LIN {X 0,Y 418.254,Z 60.388,A -85,B 0,C 180,E1 -10209.681,E2 -10209.681} C_VEL
LIN {X 0,Y 418.228,Z 60.388,A -85,B 0,C 180,E1 -10212.321,E2 -10212.321} C_VEL
LIN {X 0,Y 418.234,Z 60.379,A -85,B 0,C 180,E1 -10215.108,E2 -10215.108} C_VEL
LIN {X 0,Y 418.254,Z 60.387,A -85,B 0,C 180,E1 -10217.769,E2 -10217.769} C_VEL
LIN {X 0,Y 418.266,Z 60.381,A -85,B 0,C 180,E1 -10220.616,E2 -10220.616} C_VEL
LIN {X 0,Y 418.244,Z 60.385,A -85,B 0,C 180,E1 -10223.976,E2 -10223.976} C_VEL
LIN {X 0,Y 418.255,Z 60.388,A -85,B 0,C 180,E1 -10227.156,E2 -10227.156} C_VEL
LIN {X 0,Y 418.266,Z 60.385,A -85,B 0,C 180,E1 -10230.895,E2 -10230.895} C_VEL
LIN {X 0,Y 418.269,Z 60.378,A -85,B 0,C 180,E1 -10234.096,E2 -10234.096} C_VEL
LIN {X 0,Y 418.236,Z 60.379,A -85,B 0,C 180,E1 -10237.264,E2 -10237.264} C_VEL
LIN {X 0,Y 418.314,Z 60.38,A -85,B 0,C 180,E1 -10240.366,E2 -10240.366} C_VEL
LIN {X 0,Y 418.315,Z 60.373,A -85,B 0,C 180,E1 -10243.405,E2 -10243.405} C_VEL
LIN {X 0,Y 418.343,Z 60.364,A -85,B 0,C 180,E1 -10246.999,E2 -10246.999} C_VEL
LIN {X 0,Y 418.355,Z 60.373,A -85,B 0,C 180,E1 -10250.329,E2 -10250.329} C_VEL
LIN {X 0,Y 418.485,Z 60.349,A -85,B 0,C 180,E1 -10253.249,E2 -10253.249} C_VEL
LIN {X 0,Y 418.335,Z 60.373,A -85,B 0,C 180,E1 -10255.182,E2 -10255.182} C_VEL
LIN {X 0,Y 418.539,Z 60.345,A -85,B 0,C 180,E1 -10258.076,E2 -10258.076} C_VEL
LIN {X 0,Y 418.668,Z 60.335,A -85,B 0,C 180,E1 -10260,E2 -10260} C_VEL
LIN {X 0,Y 418.498,Z 60.346,A -85,B 0,C 180,E1 -10262.888,E2 -10262.888} C_VEL
LIN {X 0,Y 418.467,Z 60.355,A -85,B 0,C 180,E1 -10266.626,E2 -10266.626} C_VEL
LIN {X 0,Y 418.337,Z 60.376,A -85,B 0,C 180,E1 -10269.672,E2 -10269.672} C_VEL
LIN {X 0,Y 418.344,Z 60.369,A -85,B 0,C 180,E1 -10273.001,E2 -10273.001} C_VEL
LIN {X 0,Y 418.31,Z 60.378,A -85,B 0,C 180,E1 -10276.736,E2 -10276.736} C_VEL
LIN {X 0,Y 418.269,Z 60.381,A -85,B 0,C 180,E1 -10279.791,E2 -10279.791} C_VEL
LIN {X 0,Y 418.23,Z 60.386,A -85,B 0,C 180,E1 -10282.737,E2 -10282.737} C_VEL
LIN {X 0,Y 418.236,Z 60.381,A -85,B 0,C 180,E1 -10285.907,E2 -10285.907} C_VEL
LIN {X 0,Y 418.259,Z 60.38,A -85,B 0,C 180,E1 -10289.163,E2 -10289.163} C_VEL
LIN {X 0,Y 418.256,Z 60.385,A -85,B 0,C 180,E1 -10292.844,E2 -10292.844} C_VEL
LIN {X 0,Y 418.242,Z 60.39,A -85,B 0,C 180,E1 -10296.238,E2 -10296.238} C_VEL
LIN {X 0,Y 418.226,Z 60.393,A -85,B 0,C 180,E1 -10299.685,E2 -10299.685} C_VEL
LIN {X 0,Y 418.212,Z 60.393,A -85,B 0,C 180,E1 -10302.319,E2 -10302.319} C_VEL
LIN {X 0,Y 418.236,Z 60.384,A -85,B 0,C 180,E1 -10305.109,E2 -10305.109} C_VEL
LIN {X 0,Y 418.223,Z 60.394,A -85,B 0,C 180,E1 -10307.765,E2 -10307.765} C_VEL
LIN {X 0,Y 418.236,Z 60.391,A -85,B 0,C 180,E1 -10311.557,E2 -10311.557} C_VEL
LIN {X 0,Y 418.252,Z 60.396,A -85,B 0,C 180,E1 -10314.274,E2 -10314.274} C_VEL
LIN {X 0,Y 420.013,Z 68.936,A -85,B 0,C 180,E1 -10316.521,E2 -10316.521} C_VEL
LIN {X 0,Y 423.496,Z 79.315,A -85,B 0,C 180,E1 -10316.909,E2 -10316.909} C_VEL
LIN {X 0,Y 425.292,Z 87.787,A -85,B 0,C 180,E1 -10317.161,E2 -10317.161} C_VEL
LIN {X 0,Y 424.004,Z 175.768,A -85,B 0,C 180,E1 -10318.7,E2 -10318.7} C_VEL
LIN {X 0,Y 423.614,Z 189.086,A -85,B 0,C 180,E1 -10319.133,E2 -10319.133} C_VEL
LIN {X 0,Y 423.144,Z 201.473,A -85,B 0,C 180,E1 -10319.732,E2 -10319.732} C_VEL
LIN {X 0,Y 422.489,Z 212.909,A -85,B 0,C 180,E1 -10320.475,E2 -10320.475} C_VEL
LIN {X 0,Y 421.694,Z 223.677,A -85,B 0,C 180,E1 -10321.371,E2 -10321.371} C_VEL
LIN {X 0,Y 420.851,Z 234.525,A -85,B 0,C 180,E1 -10322.504,E2 -10322.504} C_VEL
LIN {X 0,Y 420.131,Z 243.656,A -85,B 0,C 180,E1 -10323.686,E2 -10323.686} C_VEL
LIN {X 0,Y 419.464,Z 251.347,A -85,B 0,C 180,E1 -10324.9,E2 -10324.9} C_VEL
LIN {X 0,Y 418.82,Z 258.37,A -85,B 0,C 180,E1 -10326.251,E2 -10326.251} C_VEL
LIN {X 0,Y 418.209,Z 265.233,A -85,B 0,C 180,E1 -10327.913,E2 -10327.913} C_VEL
LIN {X 0,Y 417.874,Z 269.767,A -85,B 0,C 180,E1 -10329.318,E2 -10329.318} C_VEL
LIN {X 0,Y 417.63,Z 272.711,A -85,B 0,C 180,E1 -10330.458,E2 -10330.458} C_VEL
LIN {X 0,Y 417.272,Z 276.201,A -85,B 0,C 180,E1 -10332.352,E2 -10332.352} C_VEL
LIN {X 0,Y 417.155,Z 277.802,A -85,B 0,C 180,E1 -10333.804,E2 -10333.804} C_VEL
LIN {X 0,Y 417.051,Z 278.53,A -85,B 0,C 180,E1 -10335.359,E2 -10335.359} C_VEL
LIN {X 0,Y 417.058,Z 278.473,A -85,B 0,C 180,E1 -10336.355,E2 -10336.355} C_VEL
LIN {X 0,Y 417.135,Z 277.669,A -85,B 0,C 180,E1 -10337.744,E2 -10337.744} C_VEL
LIN {X 0,Y 417.199,Z 275.772,A -85,B 0,C 180,E1 -10339.322,E2 -10339.322} C_VEL
LIN {X 0,Y 417.368,Z 272.99,A -85,B 0,C 180,E1 -10340.795,E2 -10340.795} C_VEL
LIN {X 0,Y 417.572,Z 269.183,A -85,B 0,C 180,E1 -10342.262,E2 -10342.262} C_VEL
LIN {X 0,Y 417.695,Z 267.355,A -85,B 0,C 180,E1 -10342.846,E2 -10342.846} C_VEL
LIN {X 0,Y 417.151,Z 264.881,A -85,B 0,C 180,E1 -10343.576,E2 -10343.576} C_VEL
LIN {X 0,Y 414.523,Z 260.479,A -85,B 0,C 180,E1 -10344.746,E2 -10344.746} C_VEL
LIN {X 0,Y 411.989,Z 255.452,A -85,B 0,C 180,E1 -10345.882,E2 -10345.882} C_VEL
LIN {X 0,Y 411.602,Z 251.956,A -85,B 0,C 180,E1 -10346.549,E2 -10346.549} C_VEL
LIN {X 0,Y 412.184,Z 244.156,A -85,B 0,C 180,E1 -10347.802,E2 -10347.802} C_VEL
LIN {X 0,Y 412.878,Z 234.823,A -85,B 0,C 180,E1 -10349.025,E2 -10349.025} C_VEL
LIN {X 0,Y 413.535,Z 224.477,A -85,B 0,C 180,E1 -10350.122,E2 -10350.122} C_VEL
LIN {X 0,Y 414.222,Z 212.979,A -85,B 0,C 180,E1 -10351.094,E2 -10351.094} C_VEL
LIN {X 0,Y 414.732,Z 200.897,A -85,B 0,C 180,E1 -10351.882,E2 -10351.882} C_VEL
LIN {X 0,Y 415.104,Z 187.886,A -85,B 0,C 180,E1 -10352.502,E2 -10352.502} C_VEL
LIN {X 0,Y 415.493,Z 174.927,A -85,B 0,C 180,E1 -10352.909,E2 -10352.909} C_VEL
LIN {X 0,Y 416.383,Z 86.513,A -85,B 0,C 180,E1 -10354.459,E2 -10354.459} C_VEL
LIN {X 0,Y 412.646,Z 68.641,A -85,B 0,C 180,E1 -10354.931,E2 -10354.931} C_VEL
LIN {X 0,Y 411.478,Z 61.231,A -85,B 0,C 180,E1 -10356.805,E2 -10356.805} C_VEL
LIN {X 0,Y 411.36,Z 61.245,A -85,B 0,C 180,E1 -10358.845,E2 -10358.845} C_VEL
LIN {X 0,Y 411.289,Z 61.25,A -85,B 0,C 180,E1 -10361.833,E2 -10361.833} C_VEL
LIN {X 0,Y 411.266,Z 61.255,A -85,B 0,C 180,E1 -10364.853,E2 -10364.853} C_VEL
LIN {X 0,Y 411.256,Z 61.256,A -85,B 0,C 180,E1 -10367.915,E2 -10367.915} C_VEL
LIN {X 0,Y 411.202,Z 61.26,A -85,B 0,C 180,E1 -10371.034,E2 -10371.034} C_VEL
LIN {X 0,Y 411.225,Z 61.263,A -85,B 0,C 180,E1 -10374.216,E2 -10374.216} C_VEL
LIN {X 0,Y 411.264,Z 61.254,A -85,B 0,C 180,E1 -10377.478,E2 -10377.478} C_VEL
LIN {X 0,Y 411.194,Z 61.261,A -85,B 0,C 180,E1 -10380.848,E2 -10380.848} C_VEL
LIN {X 0,Y 411.211,Z 61.26,A -85,B 0,C 180,E1 -10384.333,E2 -10384.333} C_VEL
LIN {X 0,Y 411.206,Z 61.263,A -85,B 0,C 180,E1 -10387.973,E2 -10387.973} C_VEL
LIN {X 0,Y 411.188,Z 61.262,A -85,B 0,C 180,E1 -10390.504,E2 -10390.504} C_VEL
LIN {X 0,Y 411.178,Z 61.267,A -85,B 0,C 180,E1 -10393.133,E2 -10393.133} C_VEL
LIN {X 0,Y 411.172,Z 61.265,A -85,B 0,C 180,E1 -10395.881,E2 -10395.881} C_VEL
LIN {X 0,Y 411.167,Z 61.266,A -85,B 0,C 180,E1 -10398.772,E2 -10398.772} C_VEL
LIN {X 0,Y 411.208,Z 61.26,A -85,B 0,C 180,E1 -10401.831,E2 -10401.831} C_VEL
LIN {X 0,Y 411.214,Z 61.264,A -85,B 0,C 180,E1 -10405.121,E2 -10405.121} C_VEL
LIN {X 0,Y 411.169,Z 61.264,A -85,B 0,C 180,E1 -10408.003,E2 -10408.003} C_VEL
LIN {X 0,Y 411.221,Z 61.259,A -85,B 0,C 180,E1 -10411.41,E2 -10411.41} C_VEL
LIN {X 0,Y 411.241,Z 61.255,A -85,B 0,C 180,E1 -10413.619,E2 -10413.619} C_VEL
LIN {X 0,Y 411.207,Z 61.264,A -85,B 0,C 180,E1 -10416.852,E2 -10416.852} C_VEL
LIN {X 0,Y 411.218,Z 61.26,A -85,B 0,C 180,E1 -10420.05,E2 -10420.05} C_VEL
LIN {X 0,Y 411.266,Z 61.253,A -85,B 0,C 180,E1 -10423.131,E2 -10423.131} C_VEL
LIN {X 0,Y 411.308,Z 61.248,A -85,B 0,C 180,E1 -10426.896,E2 -10426.896} C_VEL
LIN {X 0,Y 411.295,Z 61.255,A -85,B 0,C 180,E1 -10430.161,E2 -10430.161} C_VEL
LIN {X 0,Y 411.455,Z 61.229,A -85,B 0,C 180,E1 -10433.133,E2 -10433.133} C_VEL
LIN {X 0,Y 411.31,Z 61.247,A -85,B 0,C 180,E1 -10435.099,E2 -10435.099} C_VEL
LIN {X 0,Y 411.513,Z 61.226,A -85,B 0,C 180,E1 -10438.042,E2 -10438.042} C_VEL
LIN {X 0,Y 411.642,Z 61.21,A -85,B 0,C 180,E1 -10440,E2 -10440} C_VEL
LIN {X 0,Y 411.459,Z 61.229,A -85,B 0,C 180,E1 -10442.937,E2 -10442.937} C_VEL
LIN {X 0,Y 411.468,Z 61.231,A -85,B 0,C 180,E1 -10445.882,E2 -10445.882} C_VEL
LIN {X 0,Y 411.321,Z 61.246,A -85,B 0,C 180,E1 -10448.846,E2 -10448.846} C_VEL
LIN {X 0,Y 411.286,Z 61.252,A -85,B 0,C 180,E1 -10451.833,E2 -10451.833} C_VEL
LIN {X 0,Y 411.262,Z 61.255,A -85,B 0,C 180,E1 -10454.852,E2 -10454.852} C_VEL
LIN {X 0,Y 411.252,Z 61.254,A -85,B 0,C 180,E1 -10457.915,E2 -10457.915} C_VEL
LIN {X 0,Y 411.198,Z 61.268,A -85,B 0,C 180,E1 -10461.034,E2 -10461.034} C_VEL
LIN {X 0,Y 411.214,Z 61.259,A -85,B 0,C 180,E1 -10464.216,E2 -10464.216} C_VEL
LIN {X 0,Y 411.26,Z 61.254,A -85,B 0,C 180,E1 -10467.477,E2 -10467.477} C_VEL
LIN {X 0,Y 411.191,Z 61.267,A -85,B 0,C 180,E1 -10470.847,E2 -10470.847} C_VEL
LIN {X 0,Y 411.207,Z 61.263,A -85,B 0,C 180,E1 -10474.333,E2 -10474.333} C_VEL
LIN {X 0,Y 411.193,Z 61.263,A -85,B 0,C 180,E1 -10477.974,E2 -10477.974} C_VEL
LIN {X 0,Y 411.165,Z 61.265,A -85,B 0,C 180,E1 -10481.228,E2 -10481.228} C_VEL
LIN {X 0,Y 411.177,Z 61.267,A -85,B 0,C 180,E1 -10484.49,E2 -10484.49} C_VEL
LIN {X 0,Y 411.179,Z 61.269,A -85,B 0,C 180,E1 -10488.194,E2 -10488.194} C_VEL
LIN {X 0,Y 411.219,Z 61.258,A -85,B 0,C 180,E1 -10490.776,E2 -10490.776} C_VEL
LIN {X 0,Y 411.2,Z 61.262,A -85,B 0,C 180,E1 -10494.471,E2 -10494.471} C_VEL
LIN {X 0,Y 411.209,Z 61.259,A -85,B 0,C 180,E1 -10496.873,E2 -10496.873} C_VEL
LIN {X 0,Y 411.235,Z 61.265,A -85,B 0,C 180,E1 -10500.644,E2 -10500.644} C_VEL
LIN {X 0,Y 411.341,Z 61.434,A -85,B 0,C 180,E1 -10501.802,E2 -10501.802} C_VEL
LIN {X 0,Y 413.987,Z 75.058,A -85,B 0,C 180,E1 -10504.562,E2 -10504.562} C_VEL
LIN {X 0,Y 413.755,Z 82.381,A -85,B 0,C 180,E1 -10505.942,E2 -10505.942} C_VEL
LIN {X 0,Y 412.821,Z 97.734,A -85,B 0,C 180,E1 -10508.791,E2 -10508.791} C_VEL
LIN {X 0,Y 412.211,Z 109.992,A -85,B 0,C 180,E1 -10511.05,E2 -10511.05} C_VEL
LIN {X 0,Y 415.974,Z 138.956,A -85,B 0,C 180,E1 -10511.708,E2 -10511.708} C_VEL
LIN {X 0,Y 415.109,Z 219.027,A -85,B 0,C 180,E1 -10513.114,E2 -10513.114} C_VEL
LIN {X 0,Y 414.634,Z 232.275,A -85,B 0,C 180,E1 -10513.538,E2 -10513.538} C_VEL
LIN {X 0,Y 414.065,Z 244.461,A -85,B 0,C 180,E1 -10514.116,E2 -10514.116} C_VEL
LIN {X 0,Y 413.387,Z 255.945,A -85,B 0,C 180,E1 -10514.847,E2 -10514.847} C_VEL
LIN {X 0,Y 412.615,Z 267.749,A -85,B 0,C 180,E1 -10515.827,E2 -10515.827} C_VEL
LIN {X 0,Y 411.941,Z 278.83,A -85,B 0,C 180,E1 -10516.989,E2 -10516.989} C_VEL
LIN {X 0,Y 411.354,Z 287.906,A -85,B 0,C 180,E1 -10518.169,E2 -10518.169} C_VEL
LIN {X 0,Y 410.697,Z 297.085,A -85,B 0,C 180,E1 -10519.649,E2 -10519.649} C_VEL
LIN {X 0,Y 410.339,Z 304.487,A -85,B 0,C 180,E1 -10521.132,E2 -10521.132} C_VEL
LIN {X 0,Y 410.157,Z 310.417,A -85,B 0,C 180,E1 -10522.616,E2 -10522.616} C_VEL
LIN {X 0,Y 409.977,Z 315.069,A -85,B 0,C 180,E1 -10524.096,E2 -10524.096} C_VEL
LIN {X 0,Y 410.014,Z 318.608,A -85,B 0,C 180,E1 -10525.576,E2 -10525.576} C_VEL
LIN {X 0,Y 410.08,Z 321.12,A -85,B 0,C 180,E1 -10527.053,E2 -10527.053} C_VEL
LIN {X 0,Y 410.063,Z 322.27,A -85,B 0,C 180,E1 -10528.035,E2 -10528.035} C_VEL
LIN {X 0,Y 410.037,Z 323.303,A -85,B 0,C 180,E1 -10530,E2 -10530} C_VEL
LIN {X 0,Y 410.012,Z 323.234,A -85,B 0,C 180,E1 -10530.982,E2 -10530.982} C_VEL
LIN {X 0,Y 410.045,Z 322.766,A -85,B 0,C 180,E1 -10531.964,E2 -10531.964} C_VEL
LIN {X 0,Y 410.026,Z 321.861,A -85,B 0,C 180,E1 -10532.947,E2 -10532.947} C_VEL
LIN {X 0,Y 410.003,Z 318.854,A -85,B 0,C 180,E1 -10534.916,E2 -10534.916} C_VEL
LIN {X 0,Y 409.994,Z 315.438,A -85,B 0,C 180,E1 -10536.396,E2 -10536.396} C_VEL
LIN {X 0,Y 410.227,Z 310.958,A -85,B 0,C 180,E1 -10537.877,E2 -10537.877} C_VEL
LIN {X 0,Y 410.608,Z 304.209,A -85,B 0,C 180,E1 -10539.606,E2 -10539.606} C_VEL
LIN {X 0,Y 411.136,Z 296.87,A -85,B 0,C 180,E1 -10541.087,E2 -10541.087} C_VEL
LIN {X 0,Y 411.996,Z 287.8,A -85,B 0,C 180,E1 -10542.562,E2 -10542.562} C_VEL
LIN {X 0,Y 412.696,Z 278.456,A -85,B 0,C 180,E1 -10543.792,E2 -10543.792} C_VEL
LIN {X 0,Y 413.62,Z 268.103,A -85,B 0,C 180,E1 -10544.891,E2 -10544.891} C_VEL
LIN {X 0,Y 414.521,Z 256.647,A -85,B 0,C 180,E1 -10545.866,E2 -10545.866} C_VEL
LIN {X 0,Y 415.474,Z 244.673,A -85,B 0,C 180,E1 -10546.649,E2 -10546.649} C_VEL
LIN {X 0,Y 416.291,Z 231.401,A -85,B 0,C 180,E1 -10547.279,E2 -10547.279} C_VEL
LIN {X 0,Y 416.879,Z 218.26,A -85,B 0,C 180,E1 -10547.694,E2 -10547.694} C_VEL
LIN {X 0,Y 417.89,Z 139.457,A -85,B 0,C 180,E1 -10549.1,E2 -10549.1} C_VEL
LIN {X 0,Y 415.166,Z 121.063,A -85,B 0,C 180,E1 -10549.589,E2 -10549.589} C_VEL
LIN {X 0,Y 413.053,Z 109.27,A -85,B 0,C 180,E1 -10549.946,E2 -10549.946} C_VEL
LIN {X 0,Y 414.399,Z 89.694,A -85,B 0,C 180,E1 -10553.678,E2 -10553.678} C_VEL
LIN {X 0,Y 415.147,Z 79.905,A -85,B 0,C 180,E1 -10555.574,E2 -10555.574} C_VEL
LIN {X 0,Y 413.412,Z 70.412,A -85,B 0,C 180,E1 -10557.611,E2 -10557.611} C_VEL
LIN {X 0,Y 411.248,Z 61.264,A -85,B 0,C 180,E1 -10559.708,E2 -10559.708} C_VEL
LIN {X 0,Y 411.206,Z 61.265,A -85,B 0,C 180,E1 -10563.155,E2 -10563.155} C_VEL
LIN {X 0,Y 411.195,Z 61.266,A -85,B 0,C 180,E1 -10566.553,E2 -10566.553} C_VEL
LIN {X 0,Y 411.217,Z 61.265,A -85,B 0,C 180,E1 -10569.728,E2 -10569.728} C_VEL
LIN {X 0,Y 411.172,Z 61.267,A -85,B 0,C 180,E1 -10573.133,E2 -10573.133} C_VEL
LIN {X 0,Y 411.166,Z 61.258,A -85,B 0,C 180,E1 -10575.881,E2 -10575.881} C_VEL
LIN {X 0,Y 411.198,Z 61.263,A -85,B 0,C 180,E1 -10578.766,E2 -10578.766} C_VEL
LIN {X 0,Y 411.203,Z 61.258,A -85,B 0,C 180,E1 -10582.027,E2 -10582.027} C_VEL
LIN {X 0,Y 411.204,Z 61.26,A -85,B 0,C 180,E1 -10585.666,E2 -10585.666} C_VEL
LIN {X 0,Y 411.187,Z 61.263,A -85,B 0,C 180,E1 -10589.152,E2 -10589.152} C_VEL
LIN {X 0,Y 411.256,Z 61.257,A -85,B 0,C 180,E1 -10592.522,E2 -10592.522} C_VEL
LIN {X 0,Y 411.224,Z 61.258,A -85,B 0,C 180,E1 -10595.785,E2 -10595.785} C_VEL
LIN {X 0,Y 411.2,Z 61.264,A -85,B 0,C 180,E1 -10598.966,E2 -10598.966} C_VEL
LIN {X 0,Y 411.25,Z 61.252,A -85,B 0,C 180,E1 -10602.085,E2 -10602.085} C_VEL
LIN {X 0,Y 411.257,Z 61.254,A -85,B 0,C 180,E1 -10605.147,E2 -10605.147} C_VEL
LIN {X 0,Y 411.282,Z 61.249,A -85,B 0,C 180,E1 -10608.167,E2 -10608.167} C_VEL
LIN {X 0,Y 411.437,Z 61.228,A -85,B 0,C 180,E1 -10612.189,E2 -10612.189} C_VEL
LIN {X 0,Y 411.469,Z 61.232,A -85,B 0,C 180,E1 -10614.118,E2 -10614.118} C_VEL
LIN {X 0,Y 411.508,Z 61.22,A -85,B 0,C 180,E1 -10618.043,E2 -10618.043} C_VEL
LIN {X 0,Y 411.637,Z 61.211,A -85,B 0,C 180,E1 -10620,E2 -10620} C_VEL
LIN {X 0,Y 411.455,Z 61.223,A -85,B 0,C 180,E1 -10622.938,E2 -10622.938} C_VEL
LIN {X 0,Y 411.43,Z 61.232,A -85,B 0,C 180,E1 -10626.626,E2 -10626.626} C_VEL
LIN {X 0,Y 411.316,Z 61.242,A -85,B 0,C 180,E1 -10628.846,E2 -10628.846} C_VEL
LIN {X 0,Y 411.282,Z 61.249,A -85,B 0,C 180,E1 -10631.833,E2 -10631.833} C_VEL
LIN {X 0,Y 411.258,Z 61.256,A -85,B 0,C 180,E1 -10634.853,E2 -10634.853} C_VEL
LIN {X 0,Y 411.244,Z 61.251,A -85,B 0,C 180,E1 -10637.916,E2 -10637.916} C_VEL
LIN {X 0,Y 411.195,Z 61.261,A -85,B 0,C 180,E1 -10641.035,E2 -10641.035} C_VEL
LIN {X 0,Y 411.211,Z 61.262,A -85,B 0,C 180,E1 -10644.217,E2 -10644.217} C_VEL
LIN {X 0,Y 411.206,Z 61.261,A -85,B 0,C 180,E1 -10647.482,E2 -10647.482} C_VEL
LIN {X 0,Y 411.188,Z 61.266,A -85,B 0,C 180,E1 -10650.848,E2 -10650.848} C_VEL
LIN {X 0,Y 411.204,Z 61.265,A -85,B 0,C 180,E1 -10654.334,E2 -10654.334} C_VEL
LIN {X 0,Y 411.185,Z 61.267,A -85,B 0,C 180,E1 -10657.975,E2 -10657.975} C_VEL
LIN {X 0,Y 411.15,Z 61.262,A -85,B 0,C 180,E1 -10661.227,E2 -10661.227} C_VEL
LIN {X 0,Y 411.175,Z 61.265,A -85,B 0,C 180,E1 -10664.491,E2 -10664.491} C_VEL
LIN {X 0,Y 411.163,Z 61.27,A -85,B 0,C 180,E1 -10668.193,E2 -10668.193} C_VEL
LIN {X 0,Y 411.193,Z 61.267,A -85,B 0,C 180,E1 -10671.835,E2 -10671.835} C_VEL
LIN {X 0,Y 411.208,Z 61.279,A -85,B 0,C 180,E1 -10673.945,E2 -10673.945} C_VEL
LIN {X 0,Y 412.879,Z 69.355,A -85,B 0,C 180,E1 -10676.107,E2 -10676.107} C_VEL
LIN {X 0,Y 416.705,Z 79.72,A -85,B 0,C 180,E1 -10676.529,E2 -10676.529} C_VEL
LIN {X 0,Y 418.706,Z 88.113,A -85,B 0,C 180,E1 -10676.798,E2 -10676.798} C_VEL
LIN {X 0,Y 417.369,Z 175.969,A -85,B 0,C 180,E1 -10678.357,E2 -10678.357} C_VEL
LIN {X 0,Y 416.96,Z 189.584,A -85,B 0,C 180,E1 -10678.806,E2 -10678.806} C_VEL
LIN {X 0,Y 416.486,Z 201.398,A -85,B 0,C 180,E1 -10679.385,E2 -10679.385} C_VEL
LIN {X 0,Y 415.708,Z 214.066,A -85,B 0,C 180,E1 -10680.224,E2 -10680.224} C_VEL
LIN {X 0,Y 414.814,Z 226.061,A -85,B 0,C 180,E1 -10681.266,E2 -10681.266} C_VEL
LIN {X 0,Y 414.012,Z 235.378,A -85,B 0,C 180,E1 -10682.279,E2 -10682.279} C_VEL
LIN {X 0,Y 413.236,Z 244.438,A -85,B 0,C 180,E1 -10683.485,E2 -10683.485} C_VEL
LIN {X 0,Y 412.489,Z 252.434,A -85,B 0,C 180,E1 -10684.79,E2 -10684.79} C_VEL
LIN {X 0,Y 411.723,Z 260.168,A -85,B 0,C 180,E1 -10686.351,E2 -10686.351} C_VEL
LIN {X 0,Y 411.154,Z 266.289,A -85,B 0,C 180,E1 -10687.911,E2 -10687.911} C_VEL
LIN {X 0,Y 410.79,Z 271.033,A -85,B 0,C 180,E1 -10689.469,E2 -10689.469} C_VEL
LIN {X 0,Y 410.439,Z 274.569,A -85,B 0,C 180,E1 -10691.014,E2 -10691.014} C_VEL
LIN {X 0,Y 410.239,Z 276.296,A -85,B 0,C 180,E1 -10692.04,E2 -10692.04} C_VEL
LIN {X 0,Y 410.072,Z 278.167,A -85,B 0,C 180,E1 -10693.691,E2 -10693.691} C_VEL
LIN {X 0,Y 409.981,Z 278.887,A -85,B 0,C 180,E1 -10695.1,E2 -10695.1} C_VEL
LIN {X 0,Y 409.971,Z 278.894,A -85,B 0,C 180,E1 -10696.114,E2 -10696.114} C_VEL
LIN {X 0,Y 410.049,Z 278.096,A -85,B 0,C 180,E1 -10697.676,E2 -10697.676} C_VEL
LIN {X 0,Y 410.109,Z 276.448,A -85,B 0,C 180,E1 -10699.135,E2 -10699.135} C_VEL
LIN {X 0,Y 410.261,Z 273.799,A -85,B 0,C 180,E1 -10700.634,E2 -10700.634} C_VEL
LIN {X 0,Y 410.466,Z 270.132,A -85,B 0,C 180,E1 -10702.127,E2 -10702.127} C_VEL
LIN {X 0,Y 410.757,Z 265.347,A -85,B 0,C 180,E1 -10703.615,E2 -10703.615} C_VEL
LIN {X 0,Y 411.105,Z 259.317,A -85,B 0,C 180,E1 -10705.097,E2 -10705.097} C_VEL
LIN {X 0,Y 411.602,Z 251.956,A -85,B 0,C 180,E1 -10706.549,E2 -10706.549} C_VEL
LIN {X 0,Y 411.255,Z 248.315,A -85,B 0,C 180,E1 -10707.196,E2 -10707.196} C_VEL
LIN {X 0,Y 408.925,Z 242.07,A -85,B 0,C 180,E1 -10708.223,E2 -10708.223} C_VEL
LIN {X 0,Y 406.559,Z 235.251,A -85,B 0,C 180,E1 -10709.182,E2 -10709.182} C_VEL
LIN {X 0,Y 406.156,Z 230.71,A -85,B 0,C 180,E1 -10709.715,E2 -10709.715} C_VEL
LIN {X 0,Y 406.904,Z 220.184,A -85,B 0,C 180,E1 -10710.743,E2 -10710.743} C_VEL
LIN {X 0,Y 407.488,Z 209.129,A -85,B 0,C 180,E1 -10711.606,E2 -10711.606} C_VEL
LIN {X 0,Y 408.011,Z 197.057,A -85,B 0,C 180,E1 -10712.333,E2 -10712.333} C_VEL
LIN {X 0,Y 408.334,Z 184.687,A -85,B 0,C 180,E1 -10712.868,E2 -10712.868} C_VEL
LIN {X 0,Y 408.643,Z 171.552,A -85,B 0,C 180,E1 -10713.227,E2 -10713.227} C_VEL
LIN {X 0,Y 409.561,Z 87.33,A -85,B 0,C 180,E1 -10714.714,E2 -10714.714} C_VEL
LIN {X 0,Y 406.086,Z 70.93,A -85,B 0,C 180,E1 -10715.154,E2 -10715.154} C_VEL
LIN {X 0,Y 405.504,Z 68.987,A -85,B 0,C 180,E1 -10715.221,E2 -10715.221} C_VEL
LIN {X 0,Y 404.417,Z 62.11,A -85,B 0,C 180,E1 -10716.987,E2 -10716.987} C_VEL
LIN {X 0,Y 404.263,Z 62.126,A -85,B 0,C 180,E1 -10720.012,E2 -10720.012} C_VEL
LIN {X 0,Y 404.272,Z 62.124,A -85,B 0,C 180,E1 -10723.212,E2 -10723.212} C_VEL
LIN {X 0,Y 404.221,Z 62.131,A -85,B 0,C 180,E1 -10727.007,E2 -10727.007} C_VEL
LIN {X 0,Y 404.169,Z 62.142,A -85,B 0,C 180,E1 -10730.352,E2 -10730.352} C_VEL
LIN {X 0,Y 404.168,Z 62.138,A -85,B 0,C 180,E1 -10733.575,E2 -10733.575} C_VEL
LIN {X 0,Y 404.188,Z 62.138,A -85,B 0,C 180,E1 -10735.766,E2 -10735.766} C_VEL
LIN {X 0,Y 404.2,Z 62.139,A -85,B 0,C 180,E1 -10738,E2 -10738} C_VEL
LIN {X 0,Y 404.144,Z 62.143,A -85,B 0,C 180,E1 -10741.558,E2 -10741.558} C_VEL
LIN {X 0,Y 404.19,Z 62.134,A -85,B 0,C 180,E1 -10745.016,E2 -10745.016} C_VEL
LIN {X 0,Y 404.164,Z 62.137,A -85,B 0,C 180,E1 -10748.756,E2 -10748.756} C_VEL
LIN {X 0,Y 404.128,Z 62.147,A -85,B 0,C 180,E1 -10751.6,E2 -10751.6} C_VEL
LIN {X 0,Y 404.149,Z 62.139,A -85,B 0,C 180,E1 -10754.522,E2 -10754.522} C_VEL
LIN {X 0,Y 404.14,Z 62.147,A -85,B 0,C 180,E1 -10757.295,E2 -10757.295} C_VEL
LIN {X 0,Y 404.173,Z 62.136,A -85,B 0,C 180,E1 -10759.955,E2 -10759.955} C_VEL
LIN {X 0,Y 404.14,Z 62.146,A -85,B 0,C 180,E1 -10763.125,E2 -10763.125} C_VEL
LIN {X 0,Y 404.148,Z 62.139,A -85,B 0,C 180,E1 -10766.188,E2 -10766.188} C_VEL
LIN {X 0,Y 404.149,Z 62.139,A -85,B 0,C 180,E1 -10769.715,E2 -10769.715} C_VEL
LIN {X 0,Y 404.199,Z 62.135,A -85,B 0,C 180,E1 -10773.123,E2 -10773.123} C_VEL
LIN {X 0,Y 404.18,Z 62.136,A -85,B 0,C 180,E1 -10775.334,E2 -10775.334} C_VEL
LIN {X 0,Y 404.163,Z 62.144,A -85,B 0,C 180,E1 -10778.582,E2 -10778.582} C_VEL
LIN {X 0,Y 404.213,Z 62.131,A -85,B 0,C 180,E1 -10781.762,E2 -10781.762} C_VEL
LIN {X 0,Y 404.209,Z 62.133,A -85,B 0,C 180,E1 -10784.882,E2 -10784.882} C_VEL
LIN {X 0,Y 404.259,Z 62.129,A -85,B 0,C 180,E1 -10787.958,E2 -10787.958} C_VEL
LIN {X 0,Y 404.407,Z 62.113,A -85,B 0,C 180,E1 -10792.129,E2 -10792.129} C_VEL
LIN {X 0,Y 404.422,Z 62.112,A -85,B 0,C 180,E1 -10794.015,E2 -10794.015} C_VEL
LIN {X 0,Y 404.482,Z 62.102,A -85,B 0,C 180,E1 -10798.008,E2 -10798.008} C_VEL
LIN {X 0,Y 404.612,Z 62.086,A -85,B 0,C 180,E1 -10800,E2 -10800} C_VEL
LIN {X 0,Y 404.417,Z 62.106,A -85,B 0,C 180,E1 -10802.988,E2 -10802.988} C_VEL
LIN {X 0,Y 404.415,Z 62.108,A -85,B 0,C 180,E1 -10805.985,E2 -10805.985} C_VEL
LIN {X 0,Y 404.268,Z 62.126,A -85,B 0,C 180,E1 -10809.001,E2 -10809.001} C_VEL
LIN {X 0,Y 404.258,Z 62.126,A -85,B 0,C 180,E1 -10812.041,E2 -10812.041} C_VEL
LIN {X 0,Y 404.208,Z 62.137,A -85,B 0,C 180,E1 -10815.118,E2 -10815.118} C_VEL
LIN {X 0,Y 404.211,Z 62.131,A -85,B 0,C 180,E1 -10818.238,E2 -10818.238} C_VEL
LIN {X 0,Y 404.14,Z 62.143,A -85,B 0,C 180,E1 -10821.419,E2 -10821.419} C_VEL
LIN {X 0,Y 404.172,Z 62.14,A -85,B 0,C 180,E1 -10824.666,E2 -10824.666} C_VEL
LIN {X 0,Y 404.197,Z 62.133,A -85,B 0,C 180,E1 -10827.999,E2 -10827.999} C_VEL
LIN {X 0,Y 404.141,Z 62.14,A -85,B 0,C 180,E1 -10831.558,E2 -10831.558} C_VEL
LIN {X 0,Y 404.186,Z 62.136,A -85,B 0,C 180,E1 -10835.016,E2 -10835.016} C_VEL
LIN {X 0,Y 404.152,Z 62.142,A -85,B 0,C 180,E1 -10838.757,E2 -10838.757} C_VEL
LIN {X 0,Y 404.124,Z 62.142,A -85,B 0,C 180,E1 -10841.599,E2 -10841.599} C_VEL
LIN {X 0,Y 404.147,Z 62.143,A -85,B 0,C 180,E1 -10844.522,E2 -10844.522} C_VEL
LIN {X 0,Y 404.138,Z 62.14,A -85,B 0,C 180,E1 -10847.295,E2 -10847.295} C_VEL
LIN {X 0,Y 404.171,Z 62.142,A -85,B 0,C 180,E1 -10849.955,E2 -10849.955} C_VEL
LIN {X 0,Y 404.138,Z 62.14,A -85,B 0,C 180,E1 -10853.125,E2 -10853.125} C_VEL
LIN {X 0,Y 404.147,Z 62.142,A -85,B 0,C 180,E1 -10856.188,E2 -10856.188} C_VEL
LIN {X 0,Y 404.148,Z 62.146,A -85,B 0,C 180,E1 -10859.715,E2 -10859.715} C_VEL
LIN {X 0,Y 404.276,Z 62.286,A -85,B 0,C 180,E1 -10861.582,E2 -10861.582} C_VEL
LIN {X 0,Y 406.964,Z 76.045,A -85,B 0,C 180,E1 -10864.422,E2 -10864.422} C_VEL
LIN {X 0,Y 406.898,Z 81.691,A -85,B 0,C 180,E1 -10865.51,E2 -10865.51} C_VEL
LIN {X 0,Y 405.822,Z 98.452,A -85,B 0,C 180,E1 -10868.673,E2 -10868.673} C_VEL
LIN {X 0,Y 405.242,Z 109.579,A -85,B 0,C 180,E1 -10870.761,E2 -10870.761} C_VEL
LIN {X 0,Y 409.149,Z 141.449,A -85,B 0,C 180,E1 -10871.497,E2 -10871.497} C_VEL
LIN {X 0,Y 408.22,Z 219.027,A -85,B 0,C 180,E1 -10872.885,E2 -10872.885} C_VEL
LIN {X 0,Y 407.721,Z 232.156,A -85,B 0,C 180,E1 -10873.315,E2 -10873.315} C_VEL
LIN {X 0,Y 407.117,Z 244.28,A -85,B 0,C 180,E1 -10873.901,E2 -10873.901} C_VEL
LIN {X 0,Y 406.357,Z 256.52,A -85,B 0,C 180,E1 -10874.707,E2 -10874.707} C_VEL
LIN {X 0,Y 405.588,Z 268.151,A -85,B 0,C 180,E1 -10875.704,E2 -10875.704} C_VEL
LIN {X 0,Y 404.95,Z 278.288,A -85,B 0,C 180,E1 -10876.792,E2 -10876.792} C_VEL
LIN {X 0,Y 404.333,Z 287.191,A -85,B 0,C 180,E1 -10877.96,E2 -10877.96} C_VEL
LIN {X 0,Y 403.679,Z 296.442,A -85,B 0,C 180,E1 -10879.467,E2 -10879.467} C_VEL
LIN {X 0,Y 403.288,Z 303.889,A -85,B 0,C 180,E1 -10880.976,E2 -10880.976} C_VEL
LIN {X 0,Y 403.065,Z 309.858,A -85,B 0,C 180,E1 -10882.485,E2 -10882.485} C_VEL
LIN {X 0,Y 402.898,Z 314.552,A -85,B 0,C 180,E1 -10883.992,E2 -10883.992} C_VEL
LIN {X 0,Y 402.943,Z 318.124,A -85,B 0,C 180,E1 -10885.498,E2 -10885.498} C_VEL
LIN {X 0,Y 402.978,Z 320.666,A -85,B 0,C 180,E1 -10887.001,E2 -10887.001} C_VEL
LIN {X 0,Y 402.992,Z 321.845,A -85,B 0,C 180,E1 -10888.001,E2 -10888.001} C_VEL
LIN {X 0,Y 402.958,Z 322.574,A -85,B 0,C 180,E1 -10889,E2 -10889} C_VEL
LIN {X 0,Y 402.956,Z 322.91,A -85,B 0,C 180,E1 -10890,E2 -10890} C_VEL
LIN {X 0,Y 402.973,Z 322.412,A -85,B 0,C 180,E1 -10891.999,E2 -10891.999} C_VEL
LIN {X 0,Y 402.924,Z 321.526,A -85,B 0,C 180,E1 -10892.999,E2 -10892.999} C_VEL
LIN {X 0,Y 402.909,Z 318.548,A -85,B 0,C 180,E1 -10895.003,E2 -10895.003} C_VEL
LIN {X 0,Y 402.921,Z 315.165,A -85,B 0,C 180,E1 -10896.509,E2 -10896.509} C_VEL
LIN {X 0,Y 403.168,Z 310.723,A -85,B 0,C 180,E1 -10898.016,E2 -10898.016} C_VEL
LIN {X 0,Y 403.563,Z 304.04,A -85,B 0,C 180,E1 -10899.776,E2 -10899.776} C_VEL
LIN {X 0,Y 404.14,Z 296.758,A -85,B 0,C 180,E1 -10901.282,E2 -10901.282} C_VEL
LIN {X 0,Y 405.046,Z 287.752,A -85,B 0,C 180,E1 -10902.781,E2 -10902.781} C_VEL
LIN {X 0,Y 405.805,Z 278.51,A -85,B 0,C 180,E1 -10904.031,E2 -10904.031} C_VEL
LIN {X 0,Y 406.781,Z 268.254,A -85,B 0,C 180,E1 -10905.148,E2 -10905.148} C_VEL
LIN {X 0,Y 407.728,Z 256.919,A -85,B 0,C 180,E1 -10906.137,E2 -10906.137} C_VEL
LIN {X 0,Y 408.704,Z 245.167,A -85,B 0,C 180,E1 -10906.933,E2 -10906.933} C_VEL
LIN {X 0,Y 409.551,Z 232.286,A -85,B 0,C 180,E1 -10907.572,E2 -10907.572} C_VEL
LIN {X 0,Y 410.214,Z 218.668,A -85,B 0,C 180,E1 -10908.023,E2 -10908.023} C_VEL
LIN {X 0,Y 411.316,Z 140.265,A -85,B 0,C 180,E1 -10909.45,E2 -10909.45} C_VEL
LIN {X 0,Y 408.656,Z 122.375,A -85,B 0,C 180,E1 -10909.94,E2 -10909.94} C_VEL
LIN {X 0,Y 406.168,Z 108.891,A -85,B 0,C 180,E1 -10910.355,E2 -10910.355} C_VEL
LIN {X 0,Y 407.655,Z 89.588,A -85,B 0,C 180,E1 -10914.105,E2 -10914.105} C_VEL
LIN {X 0,Y 408.295,Z 81.451,A -85,B 0,C 180,E1 -10915.71,E2 -10915.71} C_VEL
LIN {X 0,Y 406.496,Z 71.797,A -85,B 0,C 180,E1 -10917.827,E2 -10917.827} C_VEL
LIN {X 0,Y 404.164,Z 62.145,A -85,B 0,C 180,E1 -10920.095,E2 -10920.095} C_VEL
LIN {X 0,Y 404.144,Z 62.148,A -85,B 0,C 180,E1 -10923.812,E2 -10923.812} C_VEL
LIN {X 0,Y 404.139,Z 62.143,A -85,B 0,C 180,E1 -10926.875,E2 -10926.875} C_VEL
LIN {X 0,Y 404.147,Z 62.143,A -85,B 0,C 180,E1 -10930.08,E2 -10930.08} C_VEL
LIN {X 0,Y 404.151,Z 62.142,A -85,B 0,C 180,E1 -10933.083,E2 -10933.083} C_VEL
LIN {X 0,Y 404.146,Z 62.132,A -85,B 0,C 180,E1 -10935.926,E2 -10935.926} C_VEL
LIN {X 0,Y 404.15,Z 62.14,A -85,B 0,C 180,E1 -10938.639,E2 -10938.639} C_VEL
LIN {X 0,Y 404.16,Z 62.14,A -85,B 0,C 180,E1 -10941.49,E2 -10941.49} C_VEL
LIN {X 0,Y 404.184,Z 62.138,A -85,B 0,C 180,E1 -10944.984,E2 -10944.984} C_VEL
LIN {X 0,Y 404.14,Z 62.143,A -85,B 0,C 180,E1 -10948.554,E2 -10948.554} C_VEL
LIN {X 0,Y 404.193,Z 62.134,A -85,B 0,C 180,E1 -10952,E2 -10952} C_VEL
LIN {X 0,Y 404.175,Z 62.138,A -85,B 0,C 180,E1 -10955.334,E2 -10955.334} C_VEL
LIN {X 0,Y 404.139,Z 62.14,A -85,B 0,C 180,E1 -10958.581,E2 -10958.581} C_VEL
LIN {X 0,Y 404.211,Z 62.128,A -85,B 0,C 180,E1 -10961.762,E2 -10961.762} C_VEL
LIN {X 0,Y 404.204,Z 62.134,A -85,B 0,C 180,E1 -10964.882,E2 -10964.882} C_VEL
LIN {X 0,Y 404.254,Z 62.121,A -85,B 0,C 180,E1 -10967.959,E2 -10967.959} C_VEL
LIN {X 0,Y 404.381,Z 62.107,A -85,B 0,C 180,E1 -10972.008,E2 -10972.008} C_VEL
LIN {X 0,Y 404.417,Z 62.108,A -85,B 0,C 180,E1 -10974.015,E2 -10974.015} C_VEL
LIN {X 0,Y 404.477,Z 62.095,A -85,B 0,C 180,E1 -10978.009,E2 -10978.009} C_VEL
LIN {X 0,Y 404.607,Z 62.087,A -85,B 0,C 180,E1 -10980,E2 -10980} C_VEL
LIN {X 0,Y 404.413,Z 62.1,A -85,B 0,C 180,E1 -10982.989,E2 -10982.989} C_VEL
LIN {X 0,Y 404.379,Z 62.11,A -85,B 0,C 180,E1 -10986.625,E2 -10986.625} C_VEL
LIN {X 0,Y 404.255,Z 62.127,A -85,B 0,C 180,E1 -10990.012,E2 -10990.012} C_VEL
LIN {X 0,Y 404.264,Z 62.123,A -85,B 0,C 180,E1 -10993.212,E2 -10993.212} C_VEL
LIN {X 0,Y 404.214,Z 62.13,A -85,B 0,C 180,E1 -10997.007,E2 -10997.007} C_VEL
LIN {X 0,Y 404.162,Z 62.14,A -85,B 0,C 180,E1 -11000.352,E2 -11000.352} C_VEL
LIN {X 0,Y 404.159,Z 62.139,A -85,B 0,C 180,E1 -11003.576,E2 -11003.576} C_VEL
LIN {X 0,Y 404.15,Z 62.144,A -85,B 0,C 180,E1 -11006.881,E2 -11006.881} C_VEL
LIN {X 0,Y 404.143,Z 62.142,A -85,B 0,C 180,E1 -11010.286,E2 -11010.286} C_VEL
LIN {X 0,Y 404.143,Z 62.143,A -85,B 0,C 180,E1 -11013.813,E2 -11013.813} C_VEL
LIN {X 0,Y 404.133,Z 62.144,A -85,B 0,C 180,E1 -11016.875,E2 -11016.875} C_VEL
LIN {X 0,Y 404.147,Z 62.141,A -85,B 0,C 180,E1 -11020.081,E2 -11020.081} C_VEL
LIN {X 0,Y 404.146,Z 62.144,A -85,B 0,C 180,E1 -11024.075,E2 -11024.075} C_VEL
LIN {X 0,Y 404.125,Z 62.15,A -85,B 0,C 180,E1 -11027.295,E2 -11027.295} C_VEL
LIN {X 0,Y 404.133,Z 62.146,A -85,B 0,C 180,E1 -11029.952,E2 -11029.952} C_VEL
LIN {X 0,Y 404.162,Z 62.154,A -85,B 0,C 180,E1 -11033.6,E2 -11033.6} C_VEL
LIN {X 0,Y 405.743,Z 69.691,A -85,B 0,C 180,E1 -11035.663,E2 -11035.663} C_VEL
LIN {X 0,Y 410.43,Z 81.96,A -85,B 0,C 180,E1 -11036.196,E2 -11036.196} C_VEL
LIN {X 0,Y 412.184,Z 90.236,A -85,B 0,C 180,E1 -11036.457,E2 -11036.457} C_VEL
LIN {X 0,Y 410.749,Z 176.174,A -85,B 0,C 180,E1 -11038.003,E2 -11038.003} C_VEL
LIN {X 0,Y 410.321,Z 189.289,A -85,B 0,C 180,E1 -11038.435,E2 -11038.435} C_VEL
LIN {X 0,Y 409.835,Z 201.557,A -85,B 0,C 180,E1 -11039.04,E2 -11039.04} C_VEL
LIN {X 0,Y 409.083,Z 213.561,A -85,B 0,C 180,E1 -11039.834,E2 -11039.834} C_VEL
LIN {X 0,Y 408.212,Z 224.352,A -85,B 0,C 180,E1 -11040.757,E2 -11040.757} C_VEL
LIN {X 0,Y 407.301,Z 234.833,A -85,B 0,C 180,E1 -11041.881,E2 -11041.881} C_VEL
LIN {X 0,Y 406.506,Z 243.415,A -85,B 0,C 180,E1 -11043.011,E2 -11043.011} C_VEL
LIN {X 0,Y 405.731,Z 251.712,A -85,B 0,C 180,E1 -11044.34,E2 -11044.34} C_VEL
LIN {X 0,Y 404.865,Z 259.662,A -85,B 0,C 180,E1 -11045.925,E2 -11045.925} C_VEL
LIN {X 0,Y 404.248,Z 265.957,A -85,B 0,C 180,E1 -11047.513,E2 -11047.513} C_VEL
LIN {X 0,Y 403.804,Z 270.863,A -85,B 0,C 180,E1 -11049.097,E2 -11049.097} C_VEL
LIN {X 0,Y 403.434,Z 274.549,A -85,B 0,C 180,E1 -11050.672,E2 -11050.672} C_VEL
LIN {X 0,Y 403.211,Z 276.397,A -85,B 0,C 180,E1 -11051.716,E2 -11051.716} C_VEL
LIN {X 0,Y 402.994,Z 278.534,A -85,B 0,C 180,E1 -11053.573,E2 -11053.573} C_VEL
LIN {X 0,Y 402.931,Z 279.24,A -85,B 0,C 180,E1 -11054.833,E2 -11054.833} C_VEL
LIN {X 0,Y 402.883,Z 279.316,A -85,B 0,C 180,E1 -11055.865,E2 -11055.865} C_VEL
LIN {X 0,Y 402.95,Z 278.515,A -85,B 0,C 180,E1 -11057.614,E2 -11057.614} C_VEL
LIN {X 0,Y 403.029,Z 277.12,A -85,B 0,C 180,E1 -11058.942,E2 -11058.942} C_VEL
LIN {X 0,Y 403.146,Z 274.605,A -85,B 0,C 180,E1 -11060.468,E2 -11060.468} C_VEL
LIN {X 0,Y 403.374,Z 271.072,A -85,B 0,C 180,E1 -11061.988,E2 -11061.988} C_VEL
LIN {X 0,Y 403.702,Z 265.917,A -85,B 0,C 180,E1 -11063.646,E2 -11063.646} C_VEL
LIN {X 0,Y 404.082,Z 259.447,A -85,B 0,C 180,E1 -11065.262,E2 -11065.262} C_VEL
LIN {X 0,Y 404.617,Z 251.89,A -85,B 0,C 180,E1 -11066.764,E2 -11066.764} C_VEL
LIN {X 0,Y 405.217,Z 244.153,A -85,B 0,C 180,E1 -11068.013,E2 -11068.013} C_VEL
LIN {X 0,Y 406.012,Z 233.642,A -85,B 0,C 180,E1 -11069.38,E2 -11069.38} C_VEL
LIN {X 0,Y 406.156,Z 230.71,A -85,B 0,C 180,E1 -11069.715,E2 -11069.715} C_VEL
LIN {X 0,Y 405.762,Z 226.072,A -85,B 0,C 180,E1 -11070.221,E2 -11070.221} C_VEL
LIN {X 0,Y 402.401,Z 215.107,A -85,B 0,C 180,E1 -11071.335,E2 -11071.335} C_VEL
LIN {X 0,Y 400.925,Z 208.41,A -85,B 0,C 180,E1 -11071.894,E2 -11071.894} C_VEL
LIN {X 0,Y 400.812,Z 204.798,A -85,B 0,C 180,E1 -11072.138,E2 -11072.138} C_VEL
LIN {X 0,Y 401.256,Z 192.549,A -85,B 0,C 180,E1 -11072.805,E2 -11072.805} C_VEL
LIN {X 0,Y 401.621,Z 179.562,A -85,B 0,C 180,E1 -11073.287,E2 -11073.287} C_VEL
LIN {X 0,Y 401.908,Z 161.071,A -85,B 0,C 180,E1 -11073.674,E2 -11073.674} C_VEL
LIN {X 0,Y 402.71,Z 88.172,A -85,B 0,C 180,E1 -11074.979,E2 -11074.979} C_VEL
LIN {X 0,Y 399.53,Z 73.198,A -85,B 0,C 180,E1 -11075.388,E2 -11075.388} C_VEL
LIN {X 0,Y 398.37,Z 69.344,A -85,B 0,C 180,E1 -11075.518,E2 -11075.518} C_VEL
LIN {X 0,Y 397.385,Z 62.986,A -85,B 0,C 180,E1 -11077.177,E2 -11077.177} C_VEL
LIN {X 0,Y 397.223,Z 63.004,A -85,B 0,C 180,E1 -11080.191,E2 -11080.191} C_VEL
LIN {X 0,Y 397.232,Z 63.001,A -85,B 0,C 180,E1 -11083.321,E2 -11083.321} C_VEL
LIN {X 0,Y 397.187,Z 63.006,A -85,B 0,C 180,E1 -11087.155,E2 -11087.155} C_VEL
LIN {X 0,Y 397.108,Z 63.018,A -85,B 0,C 180,E1 -11090.73,E2 -11090.73} C_VEL
LIN {X 0,Y 397.134,Z 63.018,A -85,B 0,C 180,E1 -11094.019,E2 -11094.019} C_VEL
LIN {X 0,Y 397.199,Z 63.006,A -85,B 0,C 180,E1 -11097.39,E2 -11097.39} C_VEL
LIN {X 0,Y 397.083,Z 63.019,A -85,B 0,C 180,E1 -11100.882,E2 -11100.882} C_VEL
LIN {X 0,Y 397.131,Z 63.013,A -85,B 0,C 180,E1 -11104.493,E2 -11104.493} C_VEL
LIN {X 0,Y 397.111,Z 63.016,A -85,B 0,C 180,E1 -11108.274,E2 -11108.274} C_VEL
LIN {X 0,Y 397.094,Z 63.019,A -85,B 0,C 180,E1 -11110.908,E2 -11110.908} C_VEL
LIN {X 0,Y 397.105,Z 63.02,A -85,B 0,C 180,E1 -11113.648,E2 -11113.648} C_VEL
LIN {X 0,Y 397.106,Z 63.016,A -85,B 0,C 180,E1 -11116.521,E2 -11116.521} C_VEL
LIN {X 0,Y 397.117,Z 63.015,A -85,B 0,C 180,E1 -11120.423,E2 -11120.423} C_VEL
LIN {X 0,Y 397.112,Z 63.016,A -85,B 0,C 180,E1 -11124.265,E2 -11124.265} C_VEL
LIN {X 0,Y 397.118,Z 63.019,A -85,B 0,C 180,E1 -11126.727,E2 -11126.727} C_VEL
LIN {X 0,Y 397.128,Z 63.015,A -85,B 0,C 180,E1 -11130.296,E2 -11130.296} C_VEL
LIN {X 0,Y 397.198,Z 63.01,A -85,B 0,C 180,E1 -11132.61,E2 -11132.61} C_VEL
LIN {X 0,Y 397.136,Z 63.013,A -85,B 0,C 180,E1 -11135.982,E2 -11135.982} C_VEL
LIN {X 0,Y 397.142,Z 63.012,A -85,B 0,C 180,E1 -11139.704,E2 -11139.704} C_VEL
LIN {X 0,Y 397.185,Z 63.008,A -85,B 0,C 180,E1 -11142.845,E2 -11142.845} C_VEL
LIN {X 0,Y 397.231,Z 63.003,A -85,B 0,C 180,E1 -11146.702,E2 -11146.702} C_VEL
LIN {X 0,Y 397.22,Z 63.005,A -85,B 0,C 180,E1 -11149.809,E2 -11149.809} C_VEL
LIN {X 0,Y 397.352,Z 62.986,A -85,B 0,C 180,E1 -11152.888,E2 -11152.888} C_VEL
LIN {X 0,Y 397.254,Z 62.998,A -85,B 0,C 180,E1 -11154.925,E2 -11154.925} C_VEL
LIN {X 0,Y 397.451,Z 62.979,A -85,B 0,C 180,E1 -11157.973,E2 -11157.973} C_VEL
LIN {X 0,Y 397.581,Z 62.961,A -85,B 0,C 180,E1 -11160,E2 -11160} C_VEL
LIN {X 0,Y 397.376,Z 62.983,A -85,B 0,C 180,E1 -11163.041,E2 -11163.041} C_VEL
LIN {X 0,Y 397.366,Z 62.985,A -85,B 0,C 180,E1 -11166.091,E2 -11166.091} C_VEL
LIN {X 0,Y 397.238,Z 63.003,A -85,B 0,C 180,E1 -11169.162,E2 -11169.162} C_VEL
LIN {X 0,Y 397.221,Z 63.002,A -85,B 0,C 180,E1 -11172.258,E2 -11172.258} C_VEL
LIN {X 0,Y 397.181,Z 63.012,A -85,B 0,C 180,E1 -11175.392,E2 -11175.392} C_VEL
LIN {X 0,Y 397.163,Z 63.01,A -85,B 0,C 180,E1 -11178.573,E2 -11178.573} C_VEL
LIN {X 0,Y 397.098,Z 63.017,A -85,B 0,C 180,E1 -11181.818,E2 -11181.818} C_VEL
LIN {X 0,Y 397.153,Z 63.011,A -85,B 0,C 180,E1 -11185.512,E2 -11185.512} C_VEL
LIN {X 0,Y 397.124,Z 63.018,A -85,B 0,C 180,E1 -11188.543,E2 -11188.543} C_VEL
LIN {X 0,Y 397.08,Z 63.021,A -85,B 0,C 180,E1 -11192.071,E2 -11192.071} C_VEL
LIN {X 0,Y 397.121,Z 63.014,A -85,B 0,C 180,E1 -11195.503,E2 -11195.503} C_VEL
LIN {X 0,Y 397.128,Z 63.016,A -85,B 0,C 180,E1 -11198.861,E2 -11198.861} C_VEL
LIN {X 0,Y 397.071,Z 63.027,A -85,B 0,C 180,E1 -11202.267,E2 -11202.267} C_VEL
LIN {X 0,Y 397.088,Z 63.018,A -85,B 0,C 180,E1 -11205.069,E2 -11205.069} C_VEL
LIN {X 0,Y 397.068,Z 63.027,A -85,B 0,C 180,E1 -11208.021,E2 -11208.021} C_VEL
LIN {X 0,Y 397.131,Z 63.013,A -85,B 0,C 180,E1 -11211.138,E2 -11211.138} C_VEL
LIN {X 0,Y 397.121,Z 63.015,A -85,B 0,C 180,E1 -11214.496,E2 -11214.496} C_VEL
LIN {X 0,Y 397.081,Z 63.024,A -85,B 0,C 180,E1 -11217.928,E2 -11217.928} C_VEL
LIN {X 0,Y 397.216,Z 63.141,A -85,B 0,C 180,E1 -11221.355,E2 -11221.355} C_VEL
LIN {X 0,Y 399.88,Z 76.732,A -85,B 0,C 180,E1 -11224.215,E2 -11224.215} C_VEL
LIN {X 0,Y 400.059,Z 80.993,A -85,B 0,C 180,E1 -11225.063,E2 -11225.063} C_VEL
LIN {X 0,Y 399.013,Z 96.362,A -85,B 0,C 180,E1 -11228.019,E2 -11228.019} C_VEL
LIN {X 0,Y 398.265,Z 109.213,A -85,B 0,C 180,E1 -11230.473,E2 -11230.473} C_VEL
LIN {X 0,Y 402.296,Z 141.482,A -85,B 0,C 180,E1 -11231.235,E2 -11231.235} C_VEL
LIN {X 0,Y 401.367,Z 217.809,A -85,B 0,C 180,E1 -11232.616,E2 -11232.616} C_VEL
LIN {X 0,Y 400.88,Z 231.226,A -85,B 0,C 180,E1 -11233.054,E2 -11233.054} C_VEL
LIN {X 0,Y 400.186,Z 244.053,A -85,B 0,C 180,E1 -11233.68,E2 -11233.68} C_VEL
LIN {X 0,Y 399.476,Z 255.45,A -85,B 0,C 180,E1 -11234.437,E2 -11234.437} C_VEL
LIN {X 0,Y 398.773,Z 265.902,A -85,B 0,C 180,E1 -11235.324,E2 -11235.324} C_VEL
LIN {X 0,Y 398.014,Z 277.082,A -85,B 0,C 180,E1 -11236.514,E2 -11236.514} C_VEL
LIN {X 0,Y 397.308,Z 286.419,A -85,B 0,C 180,E1 -11237.744,E2 -11237.744} C_VEL
LIN {X 0,Y 396.747,Z 294.377,A -85,B 0,C 180,E1 -11239.022,E2 -11239.022} C_VEL
LIN {X 0,Y 396.288,Z 302.137,A -85,B 0,C 180,E1 -11240.558,E2 -11240.558} C_VEL
LIN {X 0,Y 396.005,Z 309.288,A -85,B 0,C 180,E1 -11242.351,E2 -11242.351} C_VEL
LIN {X 0,Y 395.793,Z 314.13,A -85,B 0,C 180,E1 -11243.922,E2 -11243.922} C_VEL
LIN {X 0,Y 395.872,Z 317.634,A -85,B 0,C 180,E1 -11245.417,E2 -11245.417} C_VEL
LIN {X 0,Y 395.879,Z 320.209,A -85,B 0,C 180,E1 -11246.947,E2 -11246.947} C_VEL
LIN {X 0,Y 395.922,Z 321.414,A -85,B 0,C 180,E1 -11247.965,E2 -11247.965} C_VEL
LIN {X 0,Y 395.883,Z 322.166,A -85,B 0,C 180,E1 -11248.982,E2 -11248.982} C_VEL
LIN {X 0,Y 395.877,Z 322.517,A -85,B 0,C 180,E1 -11250,E2 -11250} C_VEL
LIN {X 0,Y 395.902,Z 322.056,A -85,B 0,C 180,E1 -11252.034,E2 -11252.034} C_VEL
LIN {X 0,Y 395.822,Z 321.195,A -85,B 0,C 180,E1 -11253.053,E2 -11253.053} C_VEL
LIN {X 0,Y 395.798,Z 319.924,A -85,B 0,C 180,E1 -11254.073,E2 -11254.073} C_VEL
LIN {X 0,Y 395.778,Z 316.967,A -85,B 0,C 180,E1 -11255.737,E2 -11255.737} C_VEL
LIN {X 0,Y 396.029,Z 312.12,A -85,B 0,C 180,E1 -11257.648,E2 -11257.648} C_VEL
LIN {X 0,Y 396.382,Z 305.938,A -85,B 0,C 180,E1 -11259.439,E2 -11259.439} C_VEL
LIN {X 0,Y 396.897,Z 299.223,A -85,B 0,C 180,E1 -11260.973,E2 -11260.973} C_VEL
LIN {X 0,Y 397.798,Z 290.925,A -85,B 0,C 180,E1 -11262.499,E2 -11262.499} C_VEL
LIN {X 0,Y 398.576,Z 281.807,A -85,B 0,C 180,E1 -11263.856,E2 -11263.856} C_VEL
LIN {X 0,Y 399.65,Z 270.943,A -85,B 0,C 180,E1 -11265.151,E2 -11265.151} C_VEL
LIN {X 0,Y 400.665,Z 260.276,A -85,B 0,C 180,E1 -11266.168,E2 -11266.168} C_VEL
LIN {X 0,Y 401.663,Z 248.598,A -85,B 0,C 180,E1 -11267.042,E2 -11267.042} C_VEL
LIN {X 0,Y 402.692,Z 235.207,A -85,B 0,C 180,E1 -11267.783,E2 -11267.783} C_VEL
LIN {X 0,Y 403.478,Z 222.382,A -85,B 0,C 180,E1 -11268.272,E2 -11268.272} C_VEL
LIN {X 0,Y 403.875,Z 207.539,A -85,B 0,C 180,E1 -11268.607,E2 -11268.607} C_VEL
LIN {X 0,Y 404.658,Z 140.365,A -85,B 0,C 180,E1 -11269.836,E2 -11269.836} C_VEL
LIN {X 0,Y 401.762,Z 121.305,A -85,B 0,C 180,E1 -11270.376,E2 -11270.376} C_VEL
LIN {X 0,Y 399.346,Z 108.477,A -85,B 0,C 180,E1 -11270.787,E2 -11270.787} C_VEL
LIN {X 0,Y 400.866,Z 89.913,A -85,B 0,C 180,E1 -11274.461,E2 -11274.461} C_VEL
LIN {X 0,Y 401.409,Z 82.511,A -85,B 0,C 180,E1 -11275.957,E2 -11275.957} C_VEL
LIN {X 0,Y 399.269,Z 71.927,A -85,B 0,C 180,E1 -11278.345,E2 -11278.345} C_VEL
LIN {X 0,Y 397.118,Z 63.02,A -85,B 0,C 180,E1 -11280.48,E2 -11280.48} C_VEL
LIN {X 0,Y 397.125,Z 63.016,A -85,B 0,C 180,E1 -11284.493,E2 -11284.493} C_VEL
LIN {X 0,Y 397.106,Z 63.02,A -85,B 0,C 180,E1 -11288.274,E2 -11288.274} C_VEL
LIN {X 0,Y 397.088,Z 63.021,A -85,B 0,C 180,E1 -11290.908,E2 -11290.908} C_VEL
LIN {X 0,Y 397.099,Z 63.022,A -85,B 0,C 180,E1 -11293.648,E2 -11293.648} C_VEL
LIN {X 0,Y 397.102,Z 63.013,A -85,B 0,C 180,E1 -11296.52,E2 -11296.52} C_VEL
LIN {X 0,Y 397.119,Z 63.016,A -85,B 0,C 180,E1 -11299.551,E2 -11299.551} C_VEL
LIN {X 0,Y 397.097,Z 63.016,A -85,B 0,C 180,E1 -11302.79,E2 -11302.79} C_VEL
LIN {X 0,Y 397.116,Z 63.013,A -85,B 0,C 180,E1 -11306.282,E2 -11306.282} C_VEL
LIN {X 0,Y 397.103,Z 63.015,A -85,B 0,C 180,E1 -11310.135,E2 -11310.135} C_VEL
LIN {X 0,Y 397.192,Z 63.007,A -85,B 0,C 180,E1 -11312.61,E2 -11312.61} C_VEL
LIN {X 0,Y 397.13,Z 63.014,A -85,B 0,C 180,E1 -11315.982,E2 -11315.982} C_VEL
LIN {X 0,Y 397.152,Z 63.011,A -85,B 0,C 180,E1 -11319.698,E2 -11319.698} C_VEL
LIN {X 0,Y 397.179,Z 63.007,A -85,B 0,C 180,E1 -11322.845,E2 -11322.845} C_VEL
LIN {X 0,Y 397.224,Z 62.996,A -85,B 0,C 180,E1 -11326.679,E2 -11326.679} C_VEL
LIN {X 0,Y 397.222,Z 63.005,A -85,B 0,C 180,E1 -11329.809,E2 -11329.809} C_VEL
LIN {X 0,Y 397.347,Z 62.981,A -85,B 0,C 180,E1 -11332.888,E2 -11332.888} C_VEL
LIN {X 0,Y 397.251,Z 62.999,A -85,B 0,C 180,E1 -11334.925,E2 -11334.925} C_VEL
LIN {X 0,Y 397.446,Z 62.971,A -85,B 0,C 180,E1 -11337.973,E2 -11337.973} C_VEL
LIN {X 0,Y 397.576,Z 62.962,A -85,B 0,C 180,E1 -11340,E2 -11340} C_VEL
LIN {X 0,Y 397.372,Z 62.977,A -85,B 0,C 180,E1 -11343.042,E2 -11343.042} C_VEL
LIN {X 0,Y 397.33,Z 62.987,A -85,B 0,C 180,E1 -11346.621,E2 -11346.621} C_VEL
LIN {X 0,Y 397.233,Z 62.999,A -85,B 0,C 180,E1 -11349.163,E2 -11349.163} C_VEL
LIN {X 0,Y 397.217,Z 62.999,A -85,B 0,C 180,E1 -11352.258,E2 -11352.258} C_VEL
LIN {X 0,Y 397.177,Z 63.011,A -85,B 0,C 180,E1 -11355.392,E2 -11355.392} C_VEL
LIN {X 0,Y 397.156,Z 63.009,A -85,B 0,C 180,E1 -11358.574,E2 -11358.574} C_VEL
LIN {X 0,Y 397.094,Z 63.012,A -85,B 0,C 180,E1 -11361.819,E2 -11361.819} C_VEL
LIN {X 0,Y 397.121,Z 63.012,A -85,B 0,C 180,E1 -11365.134,E2 -11365.134} C_VEL
LIN {X 0,Y 397.098,Z 63.019,A -85,B 0,C 180,E1 -11368.546,E2 -11368.546} C_VEL
LIN {X 0,Y 397.077,Z 63.023,A -85,B 0,C 180,E1 -11372.072,E2 -11372.072} C_VEL
LIN {X 0,Y 397.117,Z 63.013,A -85,B 0,C 180,E1 -11375.504,E2 -11375.504} C_VEL
LIN {X 0,Y 397.093,Z 63.023,A -85,B 0,C 180,E1 -11378.856,E2 -11378.856} C_VEL
LIN {X 0,Y 397.056,Z 63.027,A -85,B 0,C 180,E1 -11382.269,E2 -11382.269} C_VEL
LIN {X 0,Y 397.086,Z 63.018,A -85,B 0,C 180,E1 -11385.07,E2 -11385.07} C_VEL
LIN {X 0,Y 397.053,Z 63.03,A -85,B 0,C 180,E1 -11388.024,E2 -11388.024} C_VEL
LIN {X 0,Y 397.091,Z 63.024,A -85,B 0,C 180,E1 -11391.724,E2 -11391.724} C_VEL
LIN {X 0,Y 397.113,Z 63.071,A -85,B 0,C 180,E1 -11393.245,E2 -11393.245} C_VEL
LIN {X 0,Y 398.642,Z 70.144,A -85,B 0,C 180,E1 -11395.221,E2 -11395.221} C_VEL
LIN {X 0,Y 404.22,Z 84.484,A -85,B 0,C 180,E1 -11395.86,E2 -11395.86} C_VEL
LIN {X 0,Y 405.65,Z 90.568,A -85,B 0,C 180,E1 -11396.066,E2 -11396.066} C_VEL
LIN {X 0,Y 404.168,Z 176.609,A -85,B 0,C 180,E1 -11397.64,E2 -11397.64} C_VEL
LIN {X 0,Y 403.716,Z 189.687,A -85,B 0,C 180,E1 -11398.078,E2 -11398.078} C_VEL
LIN {X 0,Y 403.235,Z 201.26,A -85,B 0,C 180,E1 -11398.653,E2 -11398.653} C_VEL
LIN {X 0,Y 402.457,Z 213.304,A -85,B 0,C 180,E1 -11399.449,E2 -11399.449} C_VEL
LIN {X 0,Y 401.58,Z 224.05,A -85,B 0,C 180,E1 -11400.37,E2 -11400.37} C_VEL
LIN {X 0,Y 400.539,Z 235.052,A -85,B 0,C 180,E1 -11401.559,E2 -11401.559} C_VEL
LIN {X 0,Y 399.638,Z 244.24,A -85,B 0,C 180,E1 -11402.792,E2 -11402.792} C_VEL
LIN {X 0,Y 398.838,Z 252.201,A -85,B 0,C 180,E1 -11404.098,E2 -11404.098} C_VEL
LIN {X 0,Y 397.904,Z 260.318,A -85,B 0,C 180,E1 -11405.755,E2 -11405.755} C_VEL
LIN {X 0,Y 397.341,Z 265.623,A -85,B 0,C 180,E1 -11407.1,E2 -11407.1} C_VEL
LIN {X 0,Y 396.836,Z 270.686,A -85,B 0,C 180,E1 -11408.712,E2 -11408.712} C_VEL
LIN {X 0,Y 396.441,Z 274.518,A -85,B 0,C 180,E1 -11410.317,E2 -11410.317} C_VEL
LIN {X 0,Y 396.192,Z 276.467,A -85,B 0,C 180,E1 -11411.38,E2 -11411.38} C_VEL
LIN {X 0,Y 396.048,Z 277.929,A -85,B 0,C 180,E1 -11412.442,E2 -11412.442} C_VEL
LIN {X 0,Y 395.928,Z 278.941,A -85,B 0,C 180,E1 -11413.501,E2 -11413.501} C_VEL
LIN {X 0,Y 395.865,Z 279.544,A -85,B 0,C 180,E1 -11414.556,E2 -11414.556} C_VEL
LIN {X 0,Y 395.806,Z 279.735,A -85,B 0,C 180,E1 -11415.607,E2 -11415.607} C_VEL
LIN {X 0,Y 395.861,Z 278.936,A -85,B 0,C 180,E1 -11417.544,E2 -11417.544} C_VEL
LIN {X 0,Y 395.935,Z 277.758,A -85,B 0,C 180,E1 -11418.741,E2 -11418.741} C_VEL
LIN {X 0,Y 395.962,Z 276.266,A -85,B 0,C 180,E1 -11419.777,E2 -11419.777} C_VEL
LIN {X 0,Y 396.217,Z 273.203,A -85,B 0,C 180,E1 -11421.329,E2 -11421.329} C_VEL
LIN {X 0,Y 396.499,Z 268.578,A -85,B 0,C 180,E1 -11423.034,E2 -11423.034} C_VEL
LIN {X 0,Y 396.772,Z 262.812,A -85,B 0,C 180,E1 -11424.665,E2 -11424.665} C_VEL
LIN {X 0,Y 397.314,Z 255.963,A -85,B 0,C 180,E1 -11426.197,E2 -11426.197} C_VEL
LIN {X 0,Y 397.881,Z 248.973,A -85,B 0,C 180,E1 -11427.469,E2 -11427.469} C_VEL
LIN {X 0,Y 398.523,Z 240.565,A -85,B 0,C 180,E1 -11428.737,E2 -11428.737} C_VEL
LIN {X 0,Y 399.261,Z 230.186,A -85,B 0,C 180,E1 -11430,E2 -11430} C_VEL
LIN {X 0,Y 400.102,Z 218.478,A -85,B 0,C 180,E1 -11431.133,E2 -11431.133} C_VEL
LIN {X 0,Y 400.711,Z 206.811,A -85,B 0,C 180,E1 -11432.011,E2 -11432.011} C_VEL
LIN {X 0,Y 400.812,Z 204.798,A -85,B 0,C 180,E1 -11432.138,E2 -11432.138} C_VEL
LIN {X 0,Y 400.419,Z 199.411,A -85,B 0,C 180,E1 -11432.482,E2 -11432.482} C_VEL
LIN {X 0,Y 397.944,Z 190.572,A -85,B 0,C 180,E1 -11433.023,E2 -11433.023} C_VEL
LIN {X 0,Y 395.4,Z 181.51,A -85,B 0,C 180,E1 -11433.465,E2 -11433.465} C_VEL
LIN {X 0,Y 394.885,Z 175.778,A -85,B 0,C 180,E1 -11433.65,E2 -11433.65} C_VEL
LIN {X 0,Y 395.897,Z 89.048,A -85,B 0,C 180,E1 -11435.247,E2 -11435.247} C_VEL
LIN {X 0,Y 392.985,Z 75.384,A -85,B 0,C 180,E1 -11435.629,E2 -11435.629} C_VEL
LIN {X 0,Y 391.275,Z 69.648,A -85,B 0,C 180,E1 -11435.836,E2 -11435.836} C_VEL
LIN {X 0,Y 390.325,Z 63.865,A -85,B 0,C 180,E1 -11437.353,E2 -11437.353} C_VEL
LIN {X 0,Y 390.173,Z 63.884,A -85,B 0,C 180,E1 -11440.377,E2 -11440.377} C_VEL
LIN {X 0,Y 390.175,Z 63.88,A -85,B 0,C 180,E1 -11443.543,E2 -11443.543} C_VEL
LIN {X 0,Y 390.154,Z 63.882,A -85,B 0,C 180,E1 -11447.308,E2 -11447.308} C_VEL
LIN {X 0,Y 390.093,Z 63.894,A -85,B 0,C 180,E1 -11450.47,E2 -11450.47} C_VEL
LIN {X 0,Y 390.078,Z 63.892,A -85,B 0,C 180,E1 -11453.352,E2 -11453.352} C_VEL
LIN {X 0,Y 390.118,Z 63.887,A -85,B 0,C 180,E1 -11456.768,E2 -11456.768} C_VEL
LIN {X 0,Y 390.044,Z 63.898,A -85,B 0,C 180,E1 -11460.3,E2 -11460.3} C_VEL
LIN {X 0,Y 390.073,Z 63.896,A -85,B 0,C 180,E1 -11464.025,E2 -11464.025} C_VEL
LIN {X 0,Y 390.05,Z 63.901,A -85,B 0,C 180,E1 -11467.551,E2 -11467.551} C_VEL
LIN {X 0,Y 390.061,Z 63.894,A -85,B 0,C 180,E1 -11470.821,E2 -11470.821} C_VEL
LIN {X 0,Y 390.059,Z 63.896,A -85,B 0,C 180,E1 -11473.886,E2 -11473.886} C_VEL
LIN {X 0,Y 390.061,Z 63.895,A -85,B 0,C 180,E1 -11476.789,E2 -11476.789} C_VEL
LIN {X 0,Y 390.06,Z 63.897,A -85,B 0,C 180,E1 -11479.56,E2 -11479.56} C_VEL
LIN {X 0,Y 390.047,Z 63.896,A -85,B 0,C 180,E1 -11482.449,E2 -11482.449} C_VEL
LIN {X 0,Y 390.072,Z 63.892,A -85,B 0,C 180,E1 -11485.975,E2 -11485.975} C_VEL
LIN {X 0,Y 390.05,Z 63.895,A -85,B 0,C 180,E1 -11489.869,E2 -11489.869} C_VEL
LIN {X 0,Y 390.117,Z 63.888,A -85,B 0,C 180,E1 -11493.232,E2 -11493.232} C_VEL
LIN {X 0,Y 390.11,Z 63.893,A -85,B 0,C 180,E1 -11496.75,E2 -11496.75} C_VEL
LIN {X 0,Y 390.107,Z 63.89,A -85,B 0,C 180,E1 -11499.983,E2 -11499.983} C_VEL
LIN {X 0,Y 390.141,Z 63.884,A -85,B 0,C 180,E1 -11503.248,E2 -11503.248} C_VEL
LIN {X 0,Y 390.197,Z 63.88,A -85,B 0,C 180,E1 -11506.561,E2 -11506.561} C_VEL
LIN {X 0,Y 390.207,Z 63.877,A -85,B 0,C 180,E1 -11510.671,E2 -11510.671} C_VEL
LIN {X 0,Y 390.327,Z 63.865,A -85,B 0,C 180,E1 -11513.798,E2 -11513.798} C_VEL
LIN {X 0,Y 390.42,Z 63.855,A -85,B 0,C 180,E1 -11517.937,E2 -11517.937} C_VEL
LIN {X 0,Y 390.55,Z 63.837,A -85,B 0,C 180,E1 -11520,E2 -11520} C_VEL
LIN {X 0,Y 390.311,Z 63.864,A -85,B 0,C 180,E1 -11523.096,E2 -11523.096} C_VEL
LIN {X 0,Y 390.319,Z 63.863,A -85,B 0,C 180,E1 -11526.202,E2 -11526.202} C_VEL
LIN {X 0,Y 390.195,Z 63.882,A -85,B 0,C 180,E1 -11529.329,E2 -11529.329} C_VEL
LIN {X 0,Y 390.173,Z 63.88,A -85,B 0,C 180,E1 -11532.483,E2 -11532.483} C_VEL
LIN {X 0,Y 390.141,Z 63.886,A -85,B 0,C 180,E1 -11535.677,E2 -11535.677} C_VEL
LIN {X 0,Y 390.107,Z 63.892,A -85,B 0,C 180,E1 -11538.922,E2 -11538.922} C_VEL
LIN {X 0,Y 390.039,Z 63.897,A -85,B 0,C 180,E1 -11542.234,E2 -11542.234} C_VEL
LIN {X 0,Y 390.119,Z 63.887,A -85,B 0,C 180,E1 -11545.743,E2 -11545.743} C_VEL
LIN {X 0,Y 390.06,Z 63.897,A -85,B 0,C 180,E1 -11549.109,E2 -11549.109} C_VEL
LIN {X 0,Y 390.044,Z 63.902,A -85,B 0,C 180,E1 -11552.721,E2 -11552.721} C_VEL
LIN {X 0,Y 390.058,Z 63.895,A -85,B 0,C 180,E1 -11555.825,E2 -11555.825} C_VEL
LIN {X 0,Y 390.069,Z 63.893,A -85,B 0,C 180,E1 -11559.218,E2 -11559.218} C_VEL
LIN {X 0,Y 390.044,Z 63.902,A -85,B 0,C 180,E1 -11562.374,E2 -11562.374} C_VEL
LIN {X 0,Y 390.046,Z 63.896,A -85,B 0,C 180,E1 -11565.354,E2 -11565.354} C_VEL
LIN {X 0,Y 390.033,Z 63.903,A -85,B 0,C 180,E1 -11568.187,E2 -11568.187} C_VEL
LIN {X 0,Y 390.091,Z 63.89,A -85,B 0,C 180,E1 -11570.907,E2 -11570.907} C_VEL
LIN {X 0,Y 390.087,Z 63.89,A -85,B 0,C 180,E1 -11574.793,E2 -11574.793} C_VEL
LIN {X 0,Y 390.034,Z 63.902,A -85,B 0,C 180,E1 -11577.875,E2 -11577.875} C_VEL
LIN {X 0,Y 390.153,Z 63.98,A -85,B 0,C 180,E1 -11581.116,E2 -11581.116} C_VEL
LIN {X 0,Y 392.824,Z 77.472,A -85,B 0,C 180,E1 -11584.015,E2 -11584.015} C_VEL
LIN {X 0,Y 393.101,Z 81.682,A -85,B 0,C 180,E1 -11584.874,E2 -11584.874} C_VEL
LIN {X 0,Y 392.028,Z 97.048,A -85,B 0,C 180,E1 -11587.884,E2 -11587.884} C_VEL
LIN {X 0,Y 391.311,Z 108.854,A -85,B 0,C 180,E1 -11590.179,E2 -11590.179} C_VEL
LIN {X 0,Y 395.456,Z 141.952,A -85,B 0,C 180,E1 -11590.973,E2 -11590.973} C_VEL
LIN {X 0,Y 394.478,Z 217.751,A -85,B 0,C 180,E1 -11592.37,E2 -11592.37} C_VEL
LIN {X 0,Y 394.002,Z 231.06,A -85,B 0,C 180,E1 -11592.816,E2 -11592.816} C_VEL
LIN {X 0,Y 393.256,Z 243.825,A -85,B 0,C 180,E1 -11593.451,E2 -11593.451} C_VEL
LIN {X 0,Y 392.471,Z 255.977,A -85,B 0,C 180,E1 -11594.285,E2 -11594.285} C_VEL
LIN {X 0,Y 391.658,Z 267.569,A -85,B 0,C 180,E1 -11595.317,E2 -11595.317} C_VEL
LIN {X 0,Y 390.925,Z 278.018,A -85,B 0,C 180,E1 -11596.484,E2 -11596.484} C_VEL
LIN {X 0,Y 390.222,Z 287.382,A -85,B 0,C 180,E1 -11597.782,E2 -11597.782} C_VEL
LIN {X 0,Y 389.537,Z 296.463,A -85,B 0,C 180,E1 -11599.343,E2 -11599.343} C_VEL
LIN {X 0,Y 389.121,Z 303.776,A -85,B 0,C 180,E1 -11600.907,E2 -11600.907} C_VEL
LIN {X 0,Y 388.921,Z 308.706,A -85,B 0,C 180,E1 -11602.21,E2 -11602.21} C_VEL
LIN {X 0,Y 388.713,Z 313.945,A -85,B 0,C 180,E1 -11603.94,E2 -11603.94} C_VEL
LIN {X 0,Y 388.799,Z 317.136,A -85,B 0,C 180,E1 -11605.334,E2 -11605.334} C_VEL
LIN {X 0,Y 388.781,Z 319.746,A -85,B 0,C 180,E1 -11606.891,E2 -11606.891} C_VEL
LIN {X 0,Y 388.852,Z 320.974,A -85,B 0,C 180,E1 -11607.928,E2 -11607.928} C_VEL
LIN {X 0,Y 388.81,Z 321.756,A -85,B 0,C 180,E1 -11608.964,E2 -11608.964} C_VEL
LIN {X 0,Y 388.801,Z 322.124,A -85,B 0,C 180,E1 -11610,E2 -11610} C_VEL
LIN {X 0,Y 388.813,Z 321.695,A -85,B 0,C 180,E1 -11612.071,E2 -11612.071} C_VEL
LIN {X 0,Y 388.722,Z 320.867,A -85,B 0,C 180,E1 -11613.109,E2 -11613.109} C_VEL
LIN {X 0,Y 388.718,Z 319.614,A -85,B 0,C 180,E1 -11614.147,E2 -11614.147} C_VEL
LIN {X 0,Y 388.726,Z 316.196,A -85,B 0,C 180,E1 -11616.078,E2 -11616.078} C_VEL
LIN {X 0,Y 388.962,Z 311.882,A -85,B 0,C 180,E1 -11617.788,E2 -11617.788} C_VEL
LIN {X 0,Y 389.338,Z 305.76,A -85,B 0,C 180,E1 -11619.611,E2 -11619.611} C_VEL
LIN {X 0,Y 389.908,Z 299.094,A -85,B 0,C 180,E1 -11621.172,E2 -11621.172} C_VEL
LIN {X 0,Y 390.846,Z 290.857,A -85,B 0,C 180,E1 -11622.725,E2 -11622.725} C_VEL
LIN {X 0,Y 391.628,Z 282.318,A -85,B 0,C 180,E1 -11624.041,E2 -11624.041} C_VEL
LIN {X 0,Y 392.693,Z 272.145,A -85,B 0,C 180,E1 -11625.306,E2 -11625.306} C_VEL
LIN {X 0,Y 393.866,Z 260.55,A -85,B 0,C 180,E1 -11626.455,E2 -11626.455} C_VEL
LIN {X 0,Y 394.899,Z 249.118,A -85,B 0,C 180,E1 -11627.343,E2 -11627.343} C_VEL
LIN {X 0,Y 395.986,Z 236.024,A -85,B 0,C 180,E1 -11628.094,E2 -11628.094} C_VEL
LIN {X 0,Y 396.837,Z 222.835,A -85,B 0,C 180,E1 -11628.622,E2 -11628.622} C_VEL
LIN {X 0,Y 397.243,Z 210.01,A -85,B 0,C 180,E1 -11628.937,E2 -11628.937} C_VEL
LIN {X 0,Y 398.13,Z 141.393,A -85,B 0,C 180,E1 -11630.212,E2 -11630.212} C_VEL
LIN {X 0,Y 395.394,Z 123.108,A -85,B 0,C 180,E1 -11630.739,E2 -11630.739} C_VEL
LIN {X 0,Y 392.546,Z 108.093,A -85,B 0,C 180,E1 -11631.228,E2 -11631.228} C_VEL
LIN {X 0,Y 394.24,Z 89.049,A -85,B 0,C 180,E1 -11635.076,E2 -11635.076} C_VEL
LIN {X 0,Y 394.509,Z 83.826,A -85,B 0,C 180,E1 -11636.162,E2 -11636.162} C_VEL
LIN {X 0,Y 392.315,Z 73.176,A -85,B 0,C 180,E1 -11638.622,E2 -11638.622} C_VEL
LIN {X 0,Y 390.043,Z 63.902,A -85,B 0,C 180,E1 -11640.898,E2 -11640.898} C_VEL
LIN {X 0,Y 390.067,Z 63.901,A -85,B 0,C 180,E1 -11644.024,E2 -11644.024} C_VEL
LIN {X 0,Y 390.045,Z 63.9,A -85,B 0,C 180,E1 -11647.551,E2 -11647.551} C_VEL
LIN {X 0,Y 390.056,Z 63.897,A -85,B 0,C 180,E1 -11650.821,E2 -11650.821} C_VEL
LIN {X 0,Y 390.053,Z 63.896,A -85,B 0,C 180,E1 -11653.886,E2 -11653.886} C_VEL
LIN {X 0,Y 390.079,Z 63.896,A -85,B 0,C 180,E1 -11657.619,E2 -11657.619} C_VEL
LIN {X 0,Y 390.093,Z 63.893,A -85,B 0,C 180,E1 -11660.908,E2 -11660.908} C_VEL
LIN {X 0,Y 390.084,Z 63.895,A -85,B 0,C 180,E1 -11664.793,E2 -11664.793} C_VEL
LIN {X 0,Y 390.029,Z 63.899,A -85,B 0,C 180,E1 -11667.875,E2 -11667.875} C_VEL
LIN {X 0,Y 390.056,Z 63.899,A -85,B 0,C 180,E1 -11670.89,E2 -11670.89} C_VEL
LIN {X 0,Y 390.117,Z 63.885,A -85,B 0,C 180,E1 -11674.256,E2 -11674.256} C_VEL
LIN {X 0,Y 390.038,Z 63.89,A -85,B 0,C 180,E1 -11677.766,E2 -11677.766} C_VEL
LIN {X 0,Y 390.114,Z 63.885,A -85,B 0,C 180,E1 -11681.079,E2 -11681.079} C_VEL
LIN {X 0,Y 390.137,Z 63.889,A -85,B 0,C 180,E1 -11684.323,E2 -11684.323} C_VEL
LIN {X 0,Y 390.168,Z 63.872,A -85,B 0,C 180,E1 -11687.517,E2 -11687.517} C_VEL
LIN {X 0,Y 390.206,Z 63.876,A -85,B 0,C 180,E1 -11690.671,E2 -11690.671} C_VEL
LIN {X 0,Y 390.322,Z 63.861,A -85,B 0,C 180,E1 -11693.798,E2 -11693.798} C_VEL
LIN {X 0,Y 390.415,Z 63.846,A -85,B 0,C 180,E1 -11697.937,E2 -11697.937} C_VEL
LIN {X 0,Y 390.545,Z 63.838,A -85,B 0,C 180,E1 -11700,E2 -11700} C_VEL
LIN {X 0,Y 390.307,Z 63.857,A -85,B 0,C 180,E1 -11703.097,E2 -11703.097} C_VEL
LIN {X 0,Y 390.285,Z 63.864,A -85,B 0,C 180,E1 -11706.614,E2 -11706.614} C_VEL
LIN {X 0,Y 390.191,Z 63.878,A -85,B 0,C 180,E1 -11709.329,E2 -11709.329} C_VEL
LIN {X 0,Y 390.169,Z 63.878,A -85,B 0,C 180,E1 -11712.483,E2 -11712.483} C_VEL
LIN {X 0,Y 390.137,Z 63.886,A -85,B 0,C 180,E1 -11715.677,E2 -11715.677} C_VEL
LIN {X 0,Y 390.101,Z 63.891,A -85,B 0,C 180,E1 -11718.923,E2 -11718.923} C_VEL
LIN {X 0,Y 390.035,Z 63.892,A -85,B 0,C 180,E1 -11722.235,E2 -11722.235} C_VEL
LIN {X 0,Y 390.082,Z 63.887,A -85,B 0,C 180,E1 -11725.733,E2 -11725.733} C_VEL
LIN {X 0,Y 390.042,Z 63.894,A -85,B 0,C 180,E1 -11729.111,E2 -11729.111} C_VEL
LIN {X 0,Y 390.042,Z 63.898,A -85,B 0,C 180,E1 -11732.722,E2 -11732.722} C_VEL
LIN {X 0,Y 390.054,Z 63.895,A -85,B 0,C 180,E1 -11735.826,E2 -11735.826} C_VEL
LIN {X 0,Y 390.037,Z 63.902,A -85,B 0,C 180,E1 -11739.213,E2 -11739.213} C_VEL
LIN {X 0,Y 390.032,Z 63.903,A -85,B 0,C 180,E1 -11742.373,E2 -11742.373} C_VEL
LIN {X 0,Y 390.043,Z 63.896,A -85,B 0,C 180,E1 -11745.355,E2 -11745.355} C_VEL
LIN {X 0,Y 390.016,Z 63.905,A -85,B 0,C 180,E1 -11748.185,E2 -11748.185} C_VEL
LIN {X 0,Y 390.057,Z 63.899,A -85,B 0,C 180,E1 -11750.904,E2 -11750.904} C_VEL
LIN {X 0,Y 390.074,Z 63.982,A -85,B 0,C 180,E1 -11752.874,E2 -11752.874} C_VEL
LIN {X 0,Y 391.523,Z 70.514,A -85,B 0,C 180,E1 -11754.742,E2 -11754.742} C_VEL
LIN {X 0,Y 397.936,Z 86.581,A -85,B 0,C 180,E1 -11755.499,E2 -11755.499} C_VEL
LIN {X 0,Y 399.085,Z 91.502,A -85,B 0,C 180,E1 -11755.67,E2 -11755.67} C_VEL
LIN {X 0,Y 397.609,Z 177.052,A -85,B 0,C 180,E1 -11757.265,E2 -11757.265} C_VEL
LIN {X 0,Y 397.122,Z 190.516,A -85,B 0,C 180,E1 -11757.727,E2 -11757.727} C_VEL
LIN {X 0,Y 396.542,Z 202.722,A -85,B 0,C 180,E1 -11758.352,E2 -11758.352} C_VEL
LIN {X 0,Y 395.735,Z 214.338,A -85,B 0,C 180,E1 -11759.15,E2 -11759.15} C_VEL
LIN {X 0,Y 394.653,Z 226.309,A -85,B 0,C 180,E1 -11760.221,E2 -11760.221} C_VEL
LIN {X 0,Y 393.712,Z 236.172,A -85,B 0,C 180,E1 -11761.332,E2 -11761.332} C_VEL
LIN {X 0,Y 392.772,Z 245.097,A -85,B 0,C 180,E1 -11762.565,E2 -11762.565} C_VEL
LIN {X 0,Y 391.82,Z 253.933,A -85,B 0,C 180,E1 -11764.081,E2 -11764.081} C_VEL
LIN {X 0,Y 390.952,Z 260.992,A -85,B 0,C 180,E1 -11765.578,E2 -11765.578} C_VEL
LIN {X 0,Y 390.25,Z 267.175,A -85,B 0,C 180,E1 -11767.221,E2 -11767.221} C_VEL
LIN {X 0,Y 389.761,Z 271.983,A -85,B 0,C 180,E1 -11768.861,E2 -11768.861} C_VEL
LIN {X 0,Y 389.327,Z 275.578,A -85,B 0,C 180,E1 -11770.491,E2 -11770.491} C_VEL
LIN {X 0,Y 389.018,Z 278.081,A -85,B 0,C 180,E1 -11772.115,E2 -11772.115} C_VEL
LIN {X 0,Y 388.85,Z 279.27,A -85,B 0,C 180,E1 -11773.32,E2 -11773.32} C_VEL
LIN {X 0,Y 388.722,Z 280.108,A -85,B 0,C 180,E1 -11775.338,E2 -11775.338} C_VEL
LIN {X 0,Y 388.734,Z 279.954,A -85,B 0,C 180,E1 -11776.407,E2 -11776.407} C_VEL
LIN {X 0,Y 388.773,Z 279.356,A -85,B 0,C 180,E1 -11777.472,E2 -11777.472} C_VEL
LIN {X 0,Y 388.825,Z 278.364,A -85,B 0,C 180,E1 -11778.532,E2 -11778.532} C_VEL
LIN {X 0,Y 388.86,Z 276.978,A -85,B 0,C 180,E1 -11779.588,E2 -11779.588} C_VEL
LIN {X 0,Y 389.113,Z 274.036,A -85,B 0,C 180,E1 -11781.169,E2 -11781.169} C_VEL
LIN {X 0,Y 389.419,Z 269.187,A -85,B 0,C 180,E1 -11783.033,E2 -11783.033} C_VEL
LIN {X 0,Y 389.751,Z 262.955,A -85,B 0,C 180,E1 -11784.828,E2 -11784.828} C_VEL
LIN {X 0,Y 390.311,Z 256.053,A -85,B 0,C 180,E1 -11786.387,E2 -11786.387} C_VEL
LIN {X 0,Y 391.062,Z 247.397,A -85,B 0,C 180,E1 -11787.941,E2 -11787.941} C_VEL
LIN {X 0,Y 391.754,Z 238.543,A -85,B 0,C 180,E1 -11789.229,E2 -11789.229} C_VEL
LIN {X 0,Y 392.45,Z 228.829,A -85,B 0,C 180,E1 -11790.385,E2 -11790.385} C_VEL
LIN {X 0,Y 393.224,Z 218.147,A -85,B 0,C 180,E1 -11791.409,E2 -11791.409} C_VEL
LIN {X 0,Y 393.849,Z 206.266,A -85,B 0,C 180,E1 -11792.299,E2 -11792.299} C_VEL
LIN {X 0,Y 394.329,Z 193.977,A -85,B 0,C 180,E1 -11792.995,E2 -11792.995} C_VEL
LIN {X 0,Y 394.746,Z 181.385,A -85,B 0,C 180,E1 -11793.494,E2 -11793.494} C_VEL
LIN {X 0,Y 394.885,Z 175.778,A -85,B 0,C 180,E1 -11793.65,E2 -11793.65} C_VEL
LIN {X 0,Y 394.351,Z 169.991,A -85,B 0,C 180,E1 -11793.806,E2 -11793.806} C_VEL
LIN {X 0,Y 389.012,Z 151.262,A -85,B 0,C 180,E1 -11794.364,E2 -11794.364} C_VEL
LIN {X 0,Y 388.453,Z 145.444,A -85,B 0,C 180,E1 -11794.493,E2 -11794.493} C_VEL
LIN {X 0,Y 389.159,Z 90.44,A -85,B 0,C 180,E1 -11795.51,E2 -11795.51} C_VEL
LIN {X 0,Y 386.376,Z 77.287,A -85,B 0,C 180,E1 -11795.885,E2 -11795.885} C_VEL
LIN {X 0,Y 384.184,Z 70.044,A -85,B 0,C 180,E1 -11796.137,E2 -11796.137} C_VEL
LIN {X 0,Y 383.287,Z 64.743,A -85,B 0,C 180,E1 -11797.56,E2 -11797.56} C_VEL
LIN {X 0,Y 383.137,Z 64.763,A -85,B 0,C 180,E1 -11800.57,E2 -11800.57} C_VEL
LIN {X 0,Y 383.132,Z 64.758,A -85,B 0,C 180,E1 -11803.796,E2 -11803.796} C_VEL
LIN {X 0,Y 383.1,Z 64.761,A -85,B 0,C 180,E1 -11807.455,E2 -11807.455} C_VEL
LIN {X 0,Y 383.034,Z 64.771,A -85,B 0,C 180,E1 -11810.647,E2 -11810.647} C_VEL
LIN {X 0,Y 383.03,Z 64.773,A -85,B 0,C 180,E1 -11813.808,E2 -11813.808} C_VEL
LIN {X 0,Y 383.085,Z 64.768,A -85,B 0,C 180,E1 -11816.123,E2 -11816.123} C_VEL
LIN {X 0,Y 382.997,Z 64.778,A -85,B 0,C 180,E1 -11819.7,E2 -11819.7} C_VEL
LIN {X 0,Y 383.016,Z 64.774,A -85,B 0,C 180,E1 -11823.4,E2 -11823.4} C_VEL
LIN {X 0,Y 383.038,Z 64.77,A -85,B 0,C 180,E1 -11826.165,E2 -11826.165} C_VEL
LIN {X 0,Y 383.014,Z 64.774,A -85,B 0,C 180,E1 -11829.958,E2 -11829.958} C_VEL
LIN {X 0,Y 383.009,Z 64.773,A -85,B 0,C 180,E1 -11832.778,E2 -11832.778} C_VEL
LIN {X 0,Y 383.001,Z 64.775,A -85,B 0,C 180,E1 -11835.789,E2 -11835.789} C_VEL
LIN {X 0,Y 382.991,Z 64.777,A -85,B 0,C 180,E1 -11838.796,E2 -11838.796} C_VEL
LIN {X 0,Y 383.003,Z 64.773,A -85,B 0,C 180,E1 -11842.096,E2 -11842.096} C_VEL
LIN {X 0,Y 383.021,Z 64.774,A -85,B 0,C 180,E1 -11845.332,E2 -11845.332} C_VEL
LIN {X 0,Y 382.986,Z 64.779,A -85,B 0,C 180,E1 -11849.081,E2 -11849.081} C_VEL
LIN {X 0,Y 383.06,Z 64.772,A -85,B 0,C 180,E1 -11852.698,E2 -11852.698} C_VEL
LIN {X 0,Y 383.055,Z 64.769,A -85,B 0,C 180,E1 -11855.04,E2 -11855.04} C_VEL
LIN {X 0,Y 383.002,Z 64.779,A -85,B 0,C 180,E1 -11858.469,E2 -11858.469} C_VEL
LIN {X 0,Y 383.066,Z 64.766,A -85,B 0,C 180,E1 -11861.826,E2 -11861.826} C_VEL
LIN {X 0,Y 383.113,Z 64.759,A -85,B 0,C 180,E1 -11865.118,E2 -11865.118} C_VEL
LIN {X 0,Y 383.1,Z 64.766,A -85,B 0,C 180,E1 -11868.358,E2 -11868.358} C_VEL
LIN {X 0,Y 383.266,Z 64.746,A -85,B 0,C 180,E1 -11871.976,E2 -11871.976} C_VEL
LIN {X 0,Y 383.199,Z 64.749,A -85,B 0,C 180,E1 -11874.738,E2 -11874.738} C_VEL
LIN {X 0,Y 383.387,Z 64.731,A -85,B 0,C 180,E1 -11877.899,E2 -11877.899} C_VEL
LIN {X 0,Y 383.52,Z 64.713,A -85,B 0,C 180,E1 -11880,E2 -11880} C_VEL
LIN {X 0,Y 383.247,Z 64.744,A -85,B 0,C 180,E1 -11883.153,E2 -11883.153} C_VEL
LIN {X 0,Y 383.274,Z 64.74,A -85,B 0,C 180,E1 -11886.316,E2 -11886.316} C_VEL
LIN {X 0,Y 383.145,Z 64.761,A -85,B 0,C 180,E1 -11889.502,E2 -11889.502} C_VEL
LIN {X 0,Y 383.138,Z 64.757,A -85,B 0,C 180,E1 -11892.716,E2 -11892.716} C_VEL
LIN {X 0,Y 383.082,Z 64.763,A -85,B 0,C 180,E1 -11895.973,E2 -11895.973} C_VEL
LIN {X 0,Y 383.062,Z 64.77,A -85,B 0,C 180,E1 -11899.283,E2 -11899.283} C_VEL
LIN {X 0,Y 382.993,Z 64.777,A -85,B 0,C 180,E1 -11902.666,E2 -11902.666} C_VEL
LIN {X 0,Y 383.081,Z 64.764,A -85,B 0,C 180,E1 -11906.123,E2 -11906.123} C_VEL
LIN {X 0,Y 382.994,Z 64.774,A -85,B 0,C 180,E1 -11909.7,E2 -11909.7} C_VEL
LIN {X 0,Y 383.005,Z 64.773,A -85,B 0,C 180,E1 -11913.401,E2 -11913.401} C_VEL
LIN {X 0,Y 383.033,Z 64.772,A -85,B 0,C 180,E1 -11916.164,E2 -11916.164} C_VEL
LIN {X 0,Y 383.009,Z 64.774,A -85,B 0,C 180,E1 -11919.958,E2 -11919.958} C_VEL
LIN {X 0,Y 383.007,Z 64.774,A -85,B 0,C 180,E1 -11922.778,E2 -11922.778} C_VEL
LIN {X 0,Y 382.998,Z 64.776,A -85,B 0,C 180,E1 -11925.789,E2 -11925.789} C_VEL
LIN {X 0,Y 382.99,Z 64.775,A -85,B 0,C 180,E1 -11928.796,E2 -11928.796} C_VEL
LIN {X 0,Y 383.001,Z 64.778,A -85,B 0,C 180,E1 -11932.096,E2 -11932.096} C_VEL
LIN {X 0,Y 383.02,Z 64.772,A -85,B 0,C 180,E1 -11935.332,E2 -11935.332} C_VEL
LIN {X 0,Y 382.985,Z 64.776,A -85,B 0,C 180,E1 -11939.081,E2 -11939.081} C_VEL
LIN {X 0,Y 383.069,Z 64.824,A -85,B 0,C 180,E1 -11940.873,E2 -11940.873} C_VEL
LIN {X 0,Y 385.716,Z 77.755,A -85,B 0,C 180,E1 -11943.714,E2 -11943.714} C_VEL
LIN {X 0,Y 386.156,Z 82.356,A -85,B 0,C 180,E1 -11944.678,E2 -11944.678} C_VEL
LIN {X 0,Y 385.048,Z 97.732,A -85,B 0,C 180,E1 -11947.744,E2 -11947.744} C_VEL
LIN {X 0,Y 384.357,Z 108.482,A -85,B 0,C 180,E1 -11949.875,E2 -11949.875} C_VEL
LIN {X 0,Y 388.634,Z 143.254,A -85,B 0,C 180,E1 -11950.722,E2 -11950.722} C_VEL
LIN {X 0,Y 387.621,Z 217.497,A -85,B 0,C 180,E1 -11952.115,E2 -11952.115} C_VEL
LIN {X 0,Y 387.123,Z 230.771,A -85,B 0,C 180,E1 -11952.569,E2 -11952.569} C_VEL
LIN {X 0,Y 386.342,Z 243.517,A -85,B 0,C 180,E1 -11953.214,E2 -11953.214} C_VEL
LIN {X 0,Y 385.636,Z 254.863,A -85,B 0,C 180,E1 -11953.999,E2 -11953.999} C_VEL
LIN {X 0,Y 384.816,Z 265.278,A -85,B 0,C 180,E1 -11954.915,E2 -11954.915} C_VEL
LIN {X 0,Y 384.06,Z 275.712,A -85,B 0,C 180,E1 -11956.059,E2 -11956.059} C_VEL
LIN {X 0,Y 383.303,Z 284.859,A -85,B 0,C 180,E1 -11957.289,E2 -11957.289} C_VEL
LIN {X 0,Y 382.741,Z 292.961,A -85,B 0,C 180,E1 -11958.615,E2 -11958.615} C_VEL
LIN {X 0,Y 382.19,Z 300.882,A -85,B 0,C 180,E1 -11960.206,E2 -11960.206} C_VEL
LIN {X 0,Y 381.938,Z 306.267,A -85,B 0,C 180,E1 -11961.535,E2 -11961.535} C_VEL
LIN {X 0,Y 381.711,Z 311.496,A -85,B 0,C 180,E1 -11963.126,E2 -11963.126} C_VEL
LIN {X 0,Y 381.666,Z 315.549,A -85,B 0,C 180,E1 -11964.717,E2 -11964.717} C_VEL
LIN {X 0,Y 381.681,Z 317.632,A -85,B 0,C 180,E1 -11965.776,E2 -11965.776} C_VEL
LIN {X 0,Y 381.783,Z 320.53,A -85,B 0,C 180,E1 -11967.89,E2 -11967.89} C_VEL
LIN {X 0,Y 381.739,Z 321.346,A -85,B 0,C 180,E1 -11968.945,E2 -11968.945} C_VEL
LIN {X 0,Y 381.728,Z 321.731,A -85,B 0,C 180,E1 -11970,E2 -11970} C_VEL
LIN {X 0,Y 381.719,Z 321.726,A -85,B 0,C 180,E1 -11971.055,E2 -11971.055} C_VEL
LIN {X 0,Y 381.727,Z 321.334,A -85,B 0,C 180,E1 -11972.11,E2 -11972.11} C_VEL
LIN {X 0,Y 381.626,Z 320.537,A -85,B 0,C 180,E1 -11973.167,E2 -11973.167} C_VEL
LIN {X 0,Y 381.639,Z 319.303,A -85,B 0,C 180,E1 -11974.224,E2 -11974.224} C_VEL
LIN {X 0,Y 381.623,Z 316.255,A -85,B 0,C 180,E1 -11976.029,E2 -11976.029} C_VEL
LIN {X 0,Y 381.885,Z 311.65,A -85,B 0,C 180,E1 -11977.933,E2 -11977.933} C_VEL
LIN {X 0,Y 382.222,Z 306.571,A -85,B 0,C 180,E1 -11979.525,E2 -11979.525} C_VEL
LIN {X 0,Y 382.792,Z 300.221,A -85,B 0,C 180,E1 -11981.115,E2 -11981.115} C_VEL
LIN {X 0,Y 383.743,Z 292.305,A -85,B 0,C 180,E1 -11982.695,E2 -11982.695} C_VEL
LIN {X 0,Y 384.591,Z 283.682,A -85,B 0,C 180,E1 -11984.101,E2 -11984.101} C_VEL
LIN {X 0,Y 385.715,Z 273.432,A -85,B 0,C 180,E1 -11985.454,E2 -11985.454} C_VEL
LIN {X 0,Y 386.948,Z 262.245,A -85,B 0,C 180,E1 -11986.622,E2 -11986.622} C_VEL
LIN {X 0,Y 388.07,Z 251.319,A -85,B 0,C 180,E1 -11987.522,E2 -11987.522} C_VEL
LIN {X 0,Y 389.088,Z 239.267,A -85,B 0,C 180,E1 -11988.29,E2 -11988.29} C_VEL
LIN {X 0,Y 390,Z 226.864,A -85,B 0,C 180,E1 -11988.859,E2 -11988.859} C_VEL
LIN {X 0,Y 390.521,Z 214.084,A -85,B 0,C 180,E1 -11989.242,E2 -11989.242} C_VEL
LIN {X 0,Y 391.671,Z 142.763,A -85,B 0,C 180,E1 -11990.59,E2 -11990.59} C_VEL
LIN {X 0,Y 388.807,Z 123.49,A -85,B 0,C 180,E1 -11991.163,E2 -11991.163} C_VEL
LIN {X 0,Y 385.767,Z 107.664,A -85,B 0,C 180,E1 -11991.7,E2 -11991.7} C_VEL
LIN {X 0,Y 387.502,Z 89.156,A -85,B 0,C 180,E1 -11995.514,E2 -11995.514} C_VEL
LIN {X 0,Y 387.611,Z 85.133,A -85,B 0,C 180,E1 -11996.373,E2 -11996.373} C_VEL
LIN {X 0,Y 385.368,Z 74.421,A -85,B 0,C 180,E1 -11998.91,E2 -11998.91} C_VEL
LIN {X 0,Y 382.982,Z 64.784,A -85,B 0,C 180,E1 -12001.34,E2 -12001.34} C_VEL
LIN {X 0,Y 383.017,Z 64.772,A -85,B 0,C 180,E1 -12004.667,E2 -12004.667} C_VEL
LIN {X 0,Y 383.001,Z 64.78,A -85,B 0,C 180,E1 -12007.904,E2 -12007.904} C_VEL
LIN {X 0,Y 382.983,Z 64.78,A -85,B 0,C 180,E1 -12011.347,E2 -12011.347} C_VEL
LIN {X 0,Y 382.994,Z 64.772,A -85,B 0,C 180,E1 -12014.303,E2 -12014.303} C_VEL
LIN {X 0,Y 383.037,Z 64.768,A -85,B 0,C 180,E1 -12017.244,E2 -12017.244} C_VEL
LIN {X 0,Y 383.02,Z 64.772,A -85,B 0,C 180,E1 -12020.412,E2 -12020.412} C_VEL
LIN {X 0,Y 383.025,Z 64.772,A -85,B 0,C 180,E1 -12024.044,E2 -12024.044} C_VEL
LIN {X 0,Y 382.984,Z 64.778,A -85,B 0,C 180,E1 -12027.578,E2 -12027.578} C_VEL
LIN {X 0,Y 382.989,Z 64.774,A -85,B 0,C 180,E1 -12030.3,E2 -12030.3} C_VEL
LIN {X 0,Y 383.054,Z 64.767,A -85,B 0,C 180,E1 -12032.698,E2 -12032.698} C_VEL
LIN {X 0,Y 383.05,Z 64.772,A -85,B 0,C 180,E1 -12035.04,E2 -12035.04} C_VEL
LIN {X 0,Y 382.996,Z 64.771,A -85,B 0,C 180,E1 -12038.469,E2 -12038.469} C_VEL
LIN {X 0,Y 383.091,Z 64.759,A -85,B 0,C 180,E1 -12041.828,E2 -12041.828} C_VEL
LIN {X 0,Y 383.107,Z 64.761,A -85,B 0,C 180,E1 -12045.118,E2 -12045.118} C_VEL
LIN {X 0,Y 383.096,Z 64.761,A -85,B 0,C 180,E1 -12048.358,E2 -12048.358} C_VEL
LIN {X 0,Y 383.261,Z 64.737,A -85,B 0,C 180,E1 -12051.976,E2 -12051.976} C_VEL
LIN {X 0,Y 383.194,Z 64.751,A -85,B 0,C 180,E1 -12054.739,E2 -12054.739} C_VEL
LIN {X 0,Y 383.382,Z 64.721,A -85,B 0,C 180,E1 -12057.899,E2 -12057.899} C_VEL
LIN {X 0,Y 383.515,Z 64.714,A -85,B 0,C 180,E1 -12060,E2 -12060} C_VEL
LIN {X 0,Y 383.243,Z 64.737,A -85,B 0,C 180,E1 -12063.154,E2 -12063.154} C_VEL
LIN {X 0,Y 383.245,Z 64.741,A -85,B 0,C 180,E1 -12066.603,E2 -12066.603} C_VEL
LIN {X 0,Y 383.141,Z 64.758,A -85,B 0,C 180,E1 -12069.503,E2 -12069.503} C_VEL
LIN {X 0,Y 383.123,Z 64.757,A -85,B 0,C 180,E1 -12073.537,E2 -12073.537} C_VEL
LIN {X 0,Y 383.092,Z 64.76,A -85,B 0,C 180,E1 -12077.07,E2 -12077.07} C_VEL
LIN {X 0,Y 383.027,Z 64.774,A -85,B 0,C 180,E1 -12080.647,E2 -12080.647} C_VEL
LIN {X 0,Y 383.018,Z 64.773,A -85,B 0,C 180,E1 -12083.809,E2 -12083.809} C_VEL
LIN {X 0,Y 383.017,Z 64.774,A -85,B 0,C 180,E1 -12087.305,E2 -12087.305} C_VEL
LIN {X 0,Y 382.981,Z 64.779,A -85,B 0,C 180,E1 -12090.919,E2 -12090.919} C_VEL
LIN {X 0,Y 383.017,Z 64.772,A -85,B 0,C 180,E1 -12094.669,E2 -12094.669} C_VEL
LIN {X 0,Y 382.993,Z 64.778,A -85,B 0,C 180,E1 -12097.903,E2 -12097.903} C_VEL
LIN {X 0,Y 382.964,Z 64.772,A -85,B 0,C 180,E1 -12101.351,E2 -12101.351} C_VEL
LIN {X 0,Y 382.994,Z 64.777,A -85,B 0,C 180,E1 -12104.304,E2 -12104.304} C_VEL
LIN {X 0,Y 383.011,Z 64.78,A -85,B 0,C 180,E1 -12107.241,E2 -12107.241} C_VEL
LIN {X 0,Y 382.985,Z 64.78,A -85,B 0,C 180,E1 -12110.42,E2 -12110.42} C_VEL
LIN {X 0,Y 383.028,Z 64.973,A -85,B 0,C 180,E1 -12112.499,E2 -12112.499} C_VEL
LIN {X 0,Y 384.43,Z 71.108,A -85,B 0,C 180,E1 -12114.26,E2 -12114.26} C_VEL
LIN {X 0,Y 391.759,Z 88.984,A -85,B 0,C 180,E1 -12115.135,E2 -12115.135} C_VEL
LIN {X 0,Y 392.652,Z 93.941,A -85,B 0,C 180,E1 -12115.294,E2 -12115.294} C_VEL
LIN {X 0,Y 391.06,Z 177.548,A -85,B 0,C 180,E1 -12116.877,E2 -12116.877} C_VEL
LIN {X 0,Y 390.546,Z 191.072,A -85,B 0,C 180,E1 -12117.351,E2 -12117.351} C_VEL
LIN {X 0,Y 389.893,Z 204.066,A -85,B 0,C 180,E1 -12118.037,E2 -12118.037} C_VEL
LIN {X 0,Y 389.011,Z 215.571,A -85,B 0,C 180,E1 -12118.859,E2 -12118.859} C_VEL
LIN {X 0,Y 387.881,Z 227.555,A -85,B 0,C 180,E1 -12119.965,E2 -12119.965} C_VEL
LIN {X 0,Y 386.765,Z 238.183,A -85,B 0,C 180,E1 -12121.215,E2 -12121.215} C_VEL
LIN {X 0,Y 385.75,Z 247.644,A -85,B 0,C 180,E1 -12122.611,E2 -12122.611} C_VEL
LIN {X 0,Y 384.819,Z 255.35,A -85,B 0,C 180,E1 -12124.004,E2 -12124.004} C_VEL
LIN {X 0,Y 383.879,Z 262.826,A -85,B 0,C 180,E1 -12125.675,E2 -12125.675} C_VEL
LIN {X 0,Y 383.14,Z 268.672,A -85,B 0,C 180,E1 -12127.344,E2 -12127.344} C_VEL
LIN {X 0,Y 382.659,Z 273.199,A -85,B 0,C 180,E1 -12129.014,E2 -12129.014} C_VEL
LIN {X 0,Y 382.215,Z 276.554,A -85,B 0,C 180,E1 -12130.672,E2 -12130.672} C_VEL
LIN {X 0,Y 381.997,Z 278.194,A -85,B 0,C 180,E1 -12131.774,E2 -12131.774} C_VEL
LIN {X 0,Y 381.797,Z 279.634,A -85,B 0,C 180,E1 -12133.178,E2 -12133.178} C_VEL
LIN {X 0,Y 381.645,Z 280.468,A -85,B 0,C 180,E1 -12135.06,E2 -12135.06} C_VEL
LIN {X 0,Y 381.631,Z 280.396,A -85,B 0,C 180,E1 -12136.149,E2 -12136.149} C_VEL
LIN {X 0,Y 381.676,Z 279.769,A -85,B 0,C 180,E1 -12137.403,E2 -12137.403} C_VEL
LIN {X 0,Y 381.767,Z 277.64,A -85,B 0,C 180,E1 -12139.392,E2 -12139.392} C_VEL
LIN {X 0,Y 381.999,Z 274.825,A -85,B 0,C 180,E1 -12141.003,E2 -12141.003} C_VEL
LIN {X 0,Y 382.253,Z 270.985,A -85,B 0,C 180,E1 -12142.606,E2 -12142.606} C_VEL
LIN {X 0,Y 382.533,Z 266.026,A -85,B 0,C 180,E1 -12144.201,E2 -12144.201} C_VEL
LIN {X 0,Y 383.049,Z 259.778,A -85,B 0,C 180,E1 -12145.792,E2 -12145.792} C_VEL
LIN {X 0,Y 383.666,Z 251.974,A -85,B 0,C 180,E1 -12147.376,E2 -12147.376} C_VEL
LIN {X 0,Y 384.473,Z 242.231,A -85,B 0,C 180,E1 -12148.953,E2 -12148.953} C_VEL
LIN {X 0,Y 385.238,Z 233.219,A -85,B 0,C 180,E1 -12150.131,E2 -12150.131} C_VEL
LIN {X 0,Y 386.048,Z 222.075,A -85,B 0,C 180,E1 -12151.304,E2 -12151.304} C_VEL
LIN {X 0,Y 386.733,Z 211.19,A -85,B 0,C 180,E1 -12152.212,E2 -12152.212} C_VEL
LIN {X 0,Y 387.284,Z 199.389,A -85,B 0,C 180,E1 -12152.978,E2 -12152.978} C_VEL
LIN {X 0,Y 387.694,Z 186.823,A -85,B 0,C 180,E1 -12153.572,E2 -12153.572} C_VEL
LIN {X 0,Y 388.073,Z 173.458,A -85,B 0,C 180,E1 -12153.968,E2 -12153.968} C_VEL
LIN {X 0,Y 388.453,Z 145.444,A -85,B 0,C 180,E1 -12154.493,E2 -12154.493} C_VEL
LIN {X 0,Y 387.918,Z 139.631,A -85,B 0,C 180,E1 -12154.626,E2 -12154.626} C_VEL
LIN {X 0,Y 382.683,Z 120.895,A -85,B 0,C 180,E1 -12155.207,E2 -12155.207} C_VEL
LIN {X 0,Y 382.062,Z 115.084,A -85,B 0,C 180,E1 -12155.347,E2 -12155.347} C_VEL
LIN {X 0,Y 382.281,Z 91.067,A -85,B 0,C 180,E1 -12155.803,E2 -12155.803} C_VEL
LIN {X 0,Y 379.86,Z 79.51,A -85,B 0,C 180,E1 -12156.137,E2 -12156.137} C_VEL
LIN {X 0,Y 377.104,Z 70.437,A -85,B 0,C 180,E1 -12156.454,E2 -12156.454} C_VEL
LIN {X 0,Y 376.254,Z 65.619,A -85,B 0,C 180,E1 -12157.8,E2 -12157.8} C_VEL
LIN {X 0,Y 376.055,Z 65.639,A -85,B 0,C 180,E1 -12161.864,E2 -12161.864} C_VEL
LIN {X 0,Y 376.064,Z 65.638,A -85,B 0,C 180,E1 -12165.168,E2 -12165.168} C_VEL
LIN {X 0,Y 376.029,Z 65.646,A -85,B 0,C 180,E1 -12168.526,E2 -12168.526} C_VEL
LIN {X 0,Y 375.963,Z 65.654,A -85,B 0,C 180,E1 -12171.955,E2 -12171.955} C_VEL
LIN {X 0,Y 376.01,Z 65.645,A -85,B 0,C 180,E1 -12175.461,E2 -12175.461} C_VEL
LIN {X 0,Y 375.966,Z 65.65,A -85,B 0,C 180,E1 -12179.08,E2 -12179.08} C_VEL
LIN {X 0,Y 375.956,Z 65.651,A -85,B 0,C 180,E1 -12182.828,E2 -12182.828} C_VEL
LIN {X 0,Y 375.963,Z 65.653,A -85,B 0,C 180,E1 -12185.415,E2 -12185.415} C_VEL
LIN {X 0,Y 375.981,Z 65.649,A -85,B 0,C 180,E1 -12188.271,E2 -12188.271} C_VEL
LIN {X 0,Y 375.939,Z 65.658,A -85,B 0,C 180,E1 -12191.601,E2 -12191.601} C_VEL
LIN {X 0,Y 375.956,Z 65.656,A -85,B 0,C 180,E1 -12195.265,E2 -12195.265} C_VEL
LIN {X 0,Y 375.943,Z 65.658,A -85,B 0,C 180,E1 -12199.133,E2 -12199.133} C_VEL
LIN {X 0,Y 375.968,Z 65.65,A -85,B 0,C 180,E1 -12201.911,E2 -12201.911} C_VEL
LIN {X 0,Y 375.983,Z 65.65,A -85,B 0,C 180,E1 -12205.332,E2 -12205.332} C_VEL
LIN {X 0,Y 375.961,Z 65.652,A -85,B 0,C 180,E1 -12208.438,E2 -12208.438} C_VEL
LIN {X 0,Y 375.986,Z 65.648,A -85,B 0,C 180,E1 -12212.14,E2 -12212.14} C_VEL
LIN {X 0,Y 376.01,Z 65.649,A -85,B 0,C 180,E1 -12214.539,E2 -12214.539} C_VEL
LIN {X 0,Y 375.971,Z 65.65,A -85,B 0,C 180,E1 -12218.046,E2 -12218.046} C_VEL
LIN {X 0,Y 376.012,Z 65.644,A -85,B 0,C 180,E1 -12221.473,E2 -12221.473} C_VEL
LIN {X 0,Y 376.061,Z 65.639,A -85,B 0,C 180,E1 -12224.832,E2 -12224.832} C_VEL
LIN {X 0,Y 376.053,Z 65.645,A -85,B 0,C 180,E1 -12228.136,E2 -12228.136} C_VEL
LIN {X 0,Y 376.221,Z 65.623,A -85,B 0,C 180,E1 -12231.919,E2 -12231.919} C_VEL
LIN {X 0,Y 376.171,Z 65.625,A -85,B 0,C 180,E1 -12234.64,E2 -12234.64} C_VEL
LIN {X 0,Y 376.353,Z 65.608,A -85,B 0,C 180,E1 -12237.859,E2 -12237.859} C_VEL
LIN {X 0,Y 376.489,Z 65.589,A -85,B 0,C 180,E1 -12240,E2 -12240} C_VEL
LIN {X 0,Y 376.185,Z 65.624,A -85,B 0,C 180,E1 -12243.213,E2 -12243.213} C_VEL
LIN {X 0,Y 376.231,Z 65.617,A -85,B 0,C 180,E1 -12246.435,E2 -12246.435} C_VEL
LIN {X 0,Y 376.116,Z 65.635,A -85,B 0,C 180,E1 -12249.681,E2 -12249.681} C_VEL
LIN {X 0,Y 376.091,Z 65.637,A -85,B 0,C 180,E1 -12253.657,E2 -12253.657} C_VEL
LIN {X 0,Y 376.045,Z 65.642,A -85,B 0,C 180,E1 -12257.607,E2 -12257.607} C_VEL
LIN {X 0,Y 375.98,Z 65.652,A -85,B 0,C 180,E1 -12260.832,E2 -12260.832} C_VEL
LIN {X 0,Y 375.989,Z 65.648,A -85,B 0,C 180,E1 -12264.282,E2 -12264.282} C_VEL
LIN {X 0,Y 376.021,Z 65.647,A -85,B 0,C 180,E1 -12266.652,E2 -12266.652} C_VEL
LIN {X 0,Y 375.966,Z 65.652,A -85,B 0,C 180,E1 -12270.312,E2 -12270.312} C_VEL
LIN {X 0,Y 375.961,Z 65.652,A -85,B 0,C 180,E1 -12274.111,E2 -12274.111} C_VEL
LIN {X 0,Y 375.954,Z 65.655,A -85,B 0,C 180,E1 -12276.741,E2 -12276.741} C_VEL
LIN {X 0,Y 375.989,Z 65.649,A -85,B 0,C 180,E1 -12279.97,E2 -12279.97} C_VEL
LIN {X 0,Y 375.931,Z 65.656,A -85,B 0,C 180,E1 -12283.766,E2 -12283.766} C_VEL
LIN {X 0,Y 375.935,Z 65.654,A -85,B 0,C 180,E1 -12286.81,E2 -12286.81} C_VEL
LIN {X 0,Y 375.964,Z 65.651,A -85,B 0,C 180,E1 -12290.537,E2 -12290.537} C_VEL
LIN {X 0,Y 375.966,Z 65.652,A -85,B 0,C 180,E1 -12293.495,E2 -12293.495} C_VEL
LIN {X 0,Y 375.964,Z 65.656,A -85,B 0,C 180,E1 -12295.889,E2 -12295.889} C_VEL
LIN {X 0,Y 375.968,Z 65.656,A -85,B 0,C 180,E1 -12299.687,E2 -12299.687} C_VEL
LIN {X 0,Y 376.047,Z 65.804,A -85,B 0,C 180,E1 -12300.659,E2 -12300.659} C_VEL
LIN {X 0,Y 378.435,Z 77.427,A -85,B 0,C 180,E1 -12303.265,E2 -12303.265} C_VEL
LIN {X 0,Y 379.187,Z 83.024,A -85,B 0,C 180,E1 -12304.473,E2 -12304.473} C_VEL
LIN {X 0,Y 378.064,Z 98.387,A -85,B 0,C 180,E1 -12307.599,E2 -12307.599} C_VEL
LIN {X 0,Y 377.37,Z 108.142,A -85,B 0,C 180,E1 -12309.56,E2 -12309.56} C_VEL
LIN {X 0,Y 381.799,Z 143.186,A -85,B 0,C 180,E1 -12310.436,E2 -12310.436} C_VEL
LIN {X 0,Y 380.765,Z 217.226,A -85,B 0,C 180,E1 -12311.852,E2 -12311.852} C_VEL
LIN {X 0,Y 380.25,Z 230.463,A -85,B 0,C 180,E1 -12312.313,E2 -12312.313} C_VEL
LIN {X 0,Y 379.451,Z 243.19,A -85,B 0,C 180,E1 -12312.97,E2 -12312.97} C_VEL
LIN {X 0,Y 378.645,Z 255.316,A -85,B 0,C 180,E1 -12313.834,E2 -12313.834} C_VEL
LIN {X 0,Y 377.805,Z 265.579,A -85,B 0,C 180,E1 -12314.766,E2 -12314.766} C_VEL
LIN {X 0,Y 376.991,Z 276.246,A -85,B 0,C 180,E1 -12315.974,E2 -12315.974} C_VEL
LIN {X 0,Y 376.182,Z 285.842,A -85,B 0,C 180,E1 -12317.319,E2 -12317.319} C_VEL
LIN {X 0,Y 375.48,Z 295.068,A -85,B 0,C 180,E1 -12318.939,E2 -12318.939} C_VEL
LIN {X 0,Y 375.019,Z 302.497,A -85,B 0,C 180,E1 -12320.562,E2 -12320.562} C_VEL
LIN {X 0,Y 374.797,Z 307.528,A -85,B 0,C 180,E1 -12321.915,E2 -12321.915} C_VEL
LIN {X 0,Y 374.566,Z 312.394,A -85,B 0,C 180,E1 -12323.536,E2 -12323.536} C_VEL
LIN {X 0,Y 374.627,Z 316.13,A -85,B 0,C 180,E1 -12325.157,E2 -12325.157} C_VEL
LIN {X 0,Y 374.59,Z 318.815,A -85,B 0,C 180,E1 -12326.773,E2 -12326.773} C_VEL
LIN {X 0,Y 374.696,Z 320.081,A -85,B 0,C 180,E1 -12327.85,E2 -12327.85} C_VEL
LIN {X 0,Y 374.671,Z 320.93,A -85,B 0,C 180,E1 -12328.925,E2 -12328.925} C_VEL
LIN {X 0,Y 374.657,Z 321.337,A -85,B 0,C 180,E1 -12330,E2 -12330} C_VEL
LIN {X 0,Y 374.651,Z 321.35,A -85,B 0,C 180,E1 -12331.074,E2 -12331.074} C_VEL
LIN {X 0,Y 374.626,Z 320.975,A -85,B 0,C 180,E1 -12332.15,E2 -12332.15} C_VEL
LIN {X 0,Y 374.534,Z 320.206,A -85,B 0,C 180,E1 -12333.227,E2 -12333.227} C_VEL
LIN {X 0,Y 374.56,Z 319.001,A -85,B 0,C 180,E1 -12334.304,E2 -12334.304} C_VEL
LIN {X 0,Y 374.569,Z 315.348,A -85,B 0,C 180,E1 -12336.464,E2 -12336.464} C_VEL
LIN {X 0,Y 374.83,Z 311.428,A -85,B 0,C 180,E1 -12338.084,E2 -12338.084} C_VEL
LIN {X 0,Y 375.18,Z 306.392,A -85,B 0,C 180,E1 -12339.705,E2 -12339.705} C_VEL
LIN {X 0,Y 375.802,Z 300.098,A -85,B 0,C 180,E1 -12341.324,E2 -12341.324} C_VEL
LIN {X 0,Y 376.807,Z 292.262,A -85,B 0,C 180,E1 -12342.933,E2 -12342.933} C_VEL
LIN {X 0,Y 377.831,Z 282.575,A -85,B 0,C 180,E1 -12344.533,E2 -12344.533} C_VEL
LIN {X 0,Y 379.018,Z 272.459,A -85,B 0,C 180,E1 -12345.872,E2 -12345.872} C_VEL
LIN {X 0,Y 380.299,Z 261.117,A -85,B 0,C 180,E1 -12347.06,E2 -12347.06} C_VEL
LIN {X 0,Y 381.422,Z 250.033,A -85,B 0,C 180,E1 -12347.976,E2 -12347.976} C_VEL
LIN {X 0,Y 382.579,Z 237.716,A -85,B 0,C 180,E1 -12348.752,E2 -12348.752} C_VEL
LIN {X 0,Y 383.531,Z 224.657,A -85,B 0,C 180,E1 -12349.328,E2 -12349.328} C_VEL
LIN {X 0,Y 384.099,Z 210.738,A -85,B 0,C 180,E1 -12349.715,E2 -12349.715} C_VEL
LIN {X 0,Y 385.077,Z 142.464,A -85,B 0,C 180,E1 -12351.031,E2 -12351.031} C_VEL
LIN {X 0,Y 382.154,Z 123.552,A -85,B 0,C 180,E1 -12351.615,E2 -12351.615} C_VEL
LIN {X 0,Y 379.004,Z 107.162,A -85,B 0,C 180,E1 -12352.204,E2 -12352.204} C_VEL
LIN {X 0,Y 380.792,Z 89.125,A -85,B 0,C 180,E1 -12355.997,E2 -12355.997} C_VEL
LIN {X 0,Y 380.49,Z 85.252,A -85,B 0,C 180,E1 -12356.879,E2 -12356.879} C_VEL
LIN {X 0,Y 378.052,Z 74.211,A -85,B 0,C 180,E1 -12359.574,E2 -12359.574} C_VEL
LIN {X 0,Y 375.96,Z 65.66,A -85,B 0,C 180,E1 -12361.797,E2 -12361.797} C_VEL
LIN {X 0,Y 375.957,Z 65.65,A -85,B 0,C 180,E1 -12365.415,E2 -12365.415} C_VEL
LIN {X 0,Y 375.975,Z 65.652,A -85,B 0,C 180,E1 -12368.271,E2 -12368.271} C_VEL
LIN {X 0,Y 375.933,Z 65.659,A -85,B 0,C 180,E1 -12371.6,E2 -12371.6} C_VEL
LIN {X 0,Y 375.925,Z 65.645,A -85,B 0,C 180,E1 -12375.268,E2 -12375.268} C_VEL
LIN {X 0,Y 375.958,Z 65.652,A -85,B 0,C 180,E1 -12378.394,E2 -12378.394} C_VEL
LIN {X 0,Y 375.976,Z 65.648,A -85,B 0,C 180,E1 -12381.728,E2 -12381.728} C_VEL
LIN {X 0,Y 375.978,Z 65.648,A -85,B 0,C 180,E1 -12385.332,E2 -12385.332} C_VEL
LIN {X 0,Y 375.955,Z 65.653,A -85,B 0,C 180,E1 -12388.438,E2 -12388.438} C_VEL
LIN {X 0,Y 375.994,Z 65.647,A -85,B 0,C 180,E1 -12392.141,E2 -12392.141} C_VEL
LIN {X 0,Y 376.004,Z 65.645,A -85,B 0,C 180,E1 -12394.539,E2 -12394.539} C_VEL
LIN {X 0,Y 375.964,Z 65.643,A -85,B 0,C 180,E1 -12398.046,E2 -12398.046} C_VEL
LIN {X 0,Y 376.027,Z 65.638,A -85,B 0,C 180,E1 -12401.474,E2 -12401.474} C_VEL
LIN {X 0,Y 376.056,Z 65.641,A -85,B 0,C 180,E1 -12404.833,E2 -12404.833} C_VEL
LIN {X 0,Y 376.048,Z 65.636,A -85,B 0,C 180,E1 -12408.137,E2 -12408.137} C_VEL
LIN {X 0,Y 376.216,Z 65.615,A -85,B 0,C 180,E1 -12411.919,E2 -12411.919} C_VEL
LIN {X 0,Y 376.167,Z 65.627,A -85,B 0,C 180,E1 -12414.64,E2 -12414.64} C_VEL
LIN {X 0,Y 376.349,Z 65.597,A -85,B 0,C 180,E1 -12417.86,E2 -12417.86} C_VEL
LIN {X 0,Y 376.484,Z 65.59,A -85,B 0,C 180,E1 -12420,E2 -12420} C_VEL
LIN {X 0,Y 376.181,Z 65.616,A -85,B 0,C 180,E1 -12423.213,E2 -12423.213} C_VEL
LIN {X 0,Y 376.211,Z 65.617,A -85,B 0,C 180,E1 -12426.589,E2 -12426.589} C_VEL
LIN {X 0,Y 376.111,Z 65.636,A -85,B 0,C 180,E1 -12429.682,E2 -12429.682} C_VEL
LIN {X 0,Y 376.087,Z 65.634,A -85,B 0,C 180,E1 -12433.658,E2 -12433.658} C_VEL
LIN {X 0,Y 376.03,Z 65.638,A -85,B 0,C 180,E1 -12437.4,E2 -12437.4} C_VEL
LIN {X 0,Y 375.976,Z 65.649,A -85,B 0,C 180,E1 -12440.833,E2 -12440.833} C_VEL
LIN {X 0,Y 375.977,Z 65.652,A -85,B 0,C 180,E1 -12444.283,E2 -12444.283} C_VEL
LIN {X 0,Y 375.963,Z 65.652,A -85,B 0,C 180,E1 -12446.657,E2 -12446.657} C_VEL
LIN {X 0,Y 375.961,Z 65.652,A -85,B 0,C 180,E1 -12450.313,E2 -12450.313} C_VEL
LIN {X 0,Y 375.959,Z 65.656,A -85,B 0,C 180,E1 -12454.112,E2 -12454.112} C_VEL
LIN {X 0,Y 375.951,Z 65.656,A -85,B 0,C 180,E1 -12456.742,E2 -12456.742} C_VEL
LIN {X 0,Y 375.967,Z 65.652,A -85,B 0,C 180,E1 -12459.967,E2 -12459.967} C_VEL
LIN {X 0,Y 375.929,Z 65.663,A -85,B 0,C 180,E1 -12463.767,E2 -12463.767} C_VEL
LIN {X 0,Y 375.934,Z 65.662,A -85,B 0,C 180,E1 -12466.811,E2 -12466.811} C_VEL
LIN {X 0,Y 375.934,Z 65.659,A -85,B 0,C 180,E1 -12470.535,E2 -12470.535} C_VEL
LIN {X 0,Y 375.953,Z 65.721,A -85,B 0,C 180,E1 -12472.038,E2 -12472.038} C_VEL
LIN {X 0,Y 377.254,Z 71.44,A -85,B 0,C 180,E1 -12473.736,E2 -12473.736} C_VEL
LIN {X 0,Y 385.612,Z 91.445,A -85,B 0,C 180,E1 -12474.76,E2 -12474.76} C_VEL
LIN {X 0,Y 386.217,Z 94.229,A -85,B 0,C 180,E1 -12474.859,E2 -12474.859} C_VEL
LIN {X 0,Y 384.532,Z 178.179,A -85,B 0,C 180,E1 -12476.476,E2 -12476.476} C_VEL
LIN {X 0,Y 384.002,Z 191.429,A -85,B 0,C 180,E1 -12476.948,E2 -12476.948} C_VEL
LIN {X 0,Y 383.314,Z 204.513,A -85,B 0,C 180,E1 -12477.65,E2 -12477.65} C_VEL
LIN {X 0,Y 382.31,Z 216.874,A -85,B 0,C 180,E1 -12478.56,E2 -12478.56} C_VEL
LIN {X 0,Y 381.128,Z 228.672,A -85,B 0,C 180,E1 -12479.683,E2 -12479.683} C_VEL
LIN {X 0,Y 379.957,Z 239.213,A -85,B 0,C 180,E1 -12480.967,E2 -12480.967} C_VEL
LIN {X 0,Y 378.885,Z 248.475,A -85,B 0,C 180,E1 -12482.372,E2 -12482.372} C_VEL
LIN {X 0,Y 377.919,Z 256.1,A -85,B 0,C 180,E1 -12483.79,E2 -12483.79} C_VEL
LIN {X 0,Y 376.92,Z 263.485,A -85,B 0,C 180,E1 -12485.489,E2 -12485.489} C_VEL
LIN {X 0,Y 376.042,Z 270.105,A -85,B 0,C 180,E1 -12487.473,E2 -12487.473} C_VEL
LIN {X 0,Y 375.505,Z 274.806,A -85,B 0,C 180,E1 -12489.36,E2 -12489.36} C_VEL
LIN {X 0,Y 374.977,Z 278.308,A -85,B 0,C 180,E1 -12491.421,E2 -12491.421} C_VEL
LIN {X 0,Y 374.735,Z 280.006,A -85,B 0,C 180,E1 -12493.037,E2 -12493.037} C_VEL
LIN {X 0,Y 374.568,Z 280.828,A -85,B 0,C 180,E1 -12494.771,E2 -12494.771} C_VEL
LIN {X 0,Y 374.559,Z 280.816,A -85,B 0,C 180,E1 -12495.882,E2 -12495.882} C_VEL
LIN {X 0,Y 374.583,Z 280.183,A -85,B 0,C 180,E1 -12497.329,E2 -12497.329} C_VEL
LIN {X 0,Y 374.681,Z 278.299,A -85,B 0,C 180,E1 -12499.189,E2 -12499.189} C_VEL
LIN {X 0,Y 374.87,Z 275.612,A -85,B 0,C 180,E1 -12500.831,E2 -12500.831} C_VEL
LIN {X 0,Y 375.147,Z 271.901,A -85,B 0,C 180,E1 -12502.465,E2 -12502.465} C_VEL
LIN {X 0,Y 375.452,Z 267.079,A -85,B 0,C 180,E1 -12504.091,E2 -12504.091} C_VEL
LIN {X 0,Y 375.961,Z 260.986,A -85,B 0,C 180,E1 -12505.712,E2 -12505.712} C_VEL
LIN {X 0,Y 376.565,Z 253.43,A -85,B 0,C 180,E1 -12507.326,E2 -12507.326} C_VEL
LIN {X 0,Y 377.23,Z 245.698,A -85,B 0,C 180,E1 -12508.666,E2 -12508.666} C_VEL
LIN {X 0,Y 378.134,Z 235.186,A -85,B 0,C 180,E1 -12510.133,E2 -12510.133} C_VEL
LIN {X 0,Y 378.993,Z 224.489,A -85,B 0,C 180,E1 -12511.329,E2 -12511.329} C_VEL
LIN {X 0,Y 379.706,Z 214.223,A -85,B 0,C 180,E1 -12512.247,E2 -12512.247} C_VEL
LIN {X 0,Y 380.338,Z 201.799,A -85,B 0,C 180,E1 -12513.108,E2 -12513.108} C_VEL
LIN {X 0,Y 380.796,Z 188.586,A -85,B 0,C 180,E1 -12513.776,E2 -12513.776} C_VEL
LIN {X 0,Y 381.205,Z 175.325,A -85,B 0,C 180,E1 -12514.203,E2 -12514.203} C_VEL
LIN {X 0,Y 382.062,Z 115.084,A -85,B 0,C 180,E1 -12515.347,E2 -12515.347} C_VEL
LIN {X 0,Y 381.451,Z 109.264,A -85,B 0,C 180,E1 -12515.486,E2 -12515.486} C_VEL
LIN {X 0,Y 378.696,Z 99.936,A -85,B 0,C 180,E1 -12515.79,E2 -12515.79} C_VEL
LIN {X 0,Y 374.935,Z 88.788,A -85,B 0,C 180,E1 -12516.181,E2 -12516.181} C_VEL
LIN {X 0,Y 374.118,Z 84.94,A -85,B 0,C 180,E1 -12516.295,E2 -12516.295} C_VEL
LIN {X 0,Y 369.98,Z 70.806,A -85,B 0,C 180,E1 -12516.785,E2 -12516.785} C_VEL
LIN {X 0,Y 369.231,Z 66.495,A -85,B 0,C 180,E1 -12517.979,E2 -12517.979} C_VEL
LIN {X 0,Y 369.01,Z 66.518,A -85,B 0,C 180,E1 -12522.093,E2 -12522.093} C_VEL
LIN {X 0,Y 369.003,Z 66.517,A -85,B 0,C 180,E1 -12525.465,E2 -12525.465} C_VEL
LIN {X 0,Y 368.987,Z 66.52,A -85,B 0,C 180,E1 -12528.893,E2 -12528.893} C_VEL
LIN {X 0,Y 368.93,Z 66.53,A -85,B 0,C 180,E1 -12532.396,E2 -12532.396} C_VEL
LIN {X 0,Y 369.005,Z 66.523,A -85,B 0,C 180,E1 -12535.98,E2 -12535.98} C_VEL
LIN {X 0,Y 368.92,Z 66.531,A -85,B 0,C 180,E1 -12539.69,E2 -12539.69} C_VEL
LIN {X 0,Y 368.903,Z 66.53,A -85,B 0,C 180,E1 -12543.044,E2 -12543.044} C_VEL
LIN {X 0,Y 368.923,Z 66.528,A -85,B 0,C 180,E1 -12546.197,E2 -12546.197} C_VEL
LIN {X 0,Y 368.909,Z 66.53,A -85,B 0,C 180,E1 -12548.953,E2 -12548.953} C_VEL
LIN {X 0,Y 368.886,Z 66.533,A -85,B 0,C 180,E1 -12552.009,E2 -12552.009} C_VEL
LIN {X 0,Y 368.929,Z 66.531,A -85,B 0,C 180,E1 -12555.183,E2 -12555.183} C_VEL
LIN {X 0,Y 368.886,Z 66.532,A -85,B 0,C 180,E1 -12558.177,E2 -12558.177} C_VEL
LIN {X 0,Y 368.912,Z 66.532,A -85,B 0,C 180,E1 -12561.359,E2 -12561.359} C_VEL
LIN {X 0,Y 368.94,Z 66.53,A -85,B 0,C 180,E1 -12565.146,E2 -12565.146} C_VEL
LIN {X 0,Y 368.932,Z 66.53,A -85,B 0,C 180,E1 -12569.046,E2 -12569.046} C_VEL
LIN {X 0,Y 368.966,Z 66.527,A -85,B 0,C 180,E1 -12572.796,E2 -12572.796} C_VEL
LIN {X 0,Y 368.948,Z 66.525,A -85,B 0,C 180,E1 -12576.113,E2 -12576.113} C_VEL
LIN {X 0,Y 368.94,Z 66.526,A -85,B 0,C 180,E1 -12579.947,E2 -12579.947} C_VEL
LIN {X 0,Y 368.979,Z 66.52,A -85,B 0,C 180,E1 -12583.398,E2 -12583.398} C_VEL
LIN {X 0,Y 369.06,Z 66.511,A -85,B 0,C 180,E1 -12586.79,E2 -12586.79} C_VEL
LIN {X 0,Y 369.07,Z 66.515,A -85,B 0,C 180,E1 -12590.131,E2 -12590.131} C_VEL
LIN {X 0,Y 369.202,Z 66.493,A -85,B 0,C 180,E1 -12593.441,E2 -12593.441} C_VEL
LIN {X 0,Y 369.318,Z 66.484,A -85,B 0,C 180,E1 -12597.819,E2 -12597.819} C_VEL
LIN {X 0,Y 369.459,Z 66.464,A -85,B 0,C 180,E1 -12600,E2 -12600} C_VEL
LIN {X 0,Y 369.318,Z 66.48,A -85,B 0,C 180,E1 -12602.181,E2 -12602.181} C_VEL
LIN {X 0,Y 369.189,Z 66.494,A -85,B 0,C 180,E1 -12606.558,E2 -12606.558} C_VEL
LIN {X 0,Y 369.066,Z 66.511,A -85,B 0,C 180,E1 -12609.868,E2 -12609.868} C_VEL
LIN {X 0,Y 369.039,Z 66.514,A -85,B 0,C 180,E1 -12613.772,E2 -12613.772} C_VEL
LIN {X 0,Y 369.003,Z 66.518,A -85,B 0,C 180,E1 -12617.768,E2 -12617.768} C_VEL
LIN {X 0,Y 368.911,Z 66.533,A -85,B 0,C 180,E1 -12621.221,E2 -12621.221} C_VEL
LIN {X 0,Y 368.955,Z 66.528,A -85,B 0,C 180,E1 -12624.775,E2 -12624.775} C_VEL
LIN {X 0,Y 368.964,Z 66.524,A -85,B 0,C 180,E1 -12627.203,E2 -12627.203} C_VEL
LIN {X 0,Y 368.92,Z 66.527,A -85,B 0,C 180,E1 -12629.69,E2 -12629.69} C_VEL
LIN {X 0,Y 368.898,Z 66.532,A -85,B 0,C 180,E1 -12633.043,E2 -12633.043} C_VEL
LIN {X 0,Y 368.918,Z 66.531,A -85,B 0,C 180,E1 -12636.197,E2 -12636.197} C_VEL
LIN {X 0,Y 368.903,Z 66.531,A -85,B 0,C 180,E1 -12638.953,E2 -12638.953} C_VEL
LIN {X 0,Y 368.883,Z 66.535,A -85,B 0,C 180,E1 -12642.009,E2 -12642.009} C_VEL
LIN {X 0,Y 368.881,Z 66.532,A -85,B 0,C 180,E1 -12645.176,E2 -12645.176} C_VEL
LIN {X 0,Y 368.885,Z 66.537,A -85,B 0,C 180,E1 -12648.177,E2 -12648.177} C_VEL
LIN {X 0,Y 368.91,Z 66.53,A -85,B 0,C 180,E1 -12651.36,E2 -12651.36} C_VEL
LIN {X 0,Y 368.938,Z 66.526,A -85,B 0,C 180,E1 -12655.146,E2 -12655.146} C_VEL
LIN {X 0,Y 368.931,Z 66.527,A -85,B 0,C 180,E1 -12659.046,E2 -12659.046} C_VEL
LIN {X 0,Y 368.967,Z 66.627,A -85,B 0,C 180,E1 -12660.399,E2 -12660.399} C_VEL
LIN {X 0,Y 371.321,Z 77.906,A -85,B 0,C 180,E1 -12662.983,E2 -12662.983} C_VEL
LIN {X 0,Y 372.214,Z 83.672,A -85,B 0,C 180,E1 -12664.26,E2 -12664.26} C_VEL
LIN {X 0,Y 371.061,Z 99.039,A -85,B 0,C 180,E1 -12667.446,E2 -12667.446} C_VEL
LIN {X 0,Y 370.429,Z 107.708,A -85,B 0,C 180,E1 -12669.23,E2 -12669.23} C_VEL
LIN {X 0,Y 374.968,Z 144.864,A -85,B 0,C 180,E1 -12670.176,E2 -12670.176} C_VEL
LIN {X 0,Y 373.917,Z 216.935,A -85,B 0,C 180,E1 -12671.578,E2 -12671.578} C_VEL
LIN {X 0,Y 373.381,Z 230.149,A -85,B 0,C 180,E1 -12672.048,E2 -12672.048} C_VEL
LIN {X 0,Y 372.558,Z 242.861,A -85,B 0,C 180,E1 -12672.715,E2 -12672.715} C_VEL
LIN {X 0,Y 371.808,Z 254.177,A -85,B 0,C 180,E1 -12673.528,E2 -12673.528} C_VEL
LIN {X 0,Y 370.89,Z 264.571,A -85,B 0,C 180,E1 -12674.475,E2 -12674.475} C_VEL
LIN {X 0,Y 369.963,Z 276.149,A -85,B 0,C 180,E1 -12675.807,E2 -12675.807} C_VEL
LIN {X 0,Y 369.205,Z 285.038,A -85,B 0,C 180,E1 -12677.075,E2 -12677.075} C_VEL
LIN {X 0,Y 368.615,Z 292.978,A -85,B 0,C 180,E1 -12678.451,E2 -12678.451} C_VEL
LIN {X 0,Y 368.046,Z 300.711,A -85,B 0,C 180,E1 -12680.104,E2 -12680.104} C_VEL
LIN {X 0,Y 367.731,Z 306.926,A -85,B 0,C 180,E1 -12681.759,E2 -12681.759} C_VEL
LIN {X 0,Y 367.49,Z 311.839,A -85,B 0,C 180,E1 -12683.411,E2 -12683.411} C_VEL
LIN {X 0,Y 367.531,Z 315.617,A -85,B 0,C 180,E1 -12685.063,E2 -12685.063} C_VEL
LIN {X 0,Y 367.499,Z 318.343,A -85,B 0,C 180,E1 -12686.711,E2 -12686.711} C_VEL
LIN {X 0,Y 367.612,Z 319.63,A -85,B 0,C 180,E1 -12687.808,E2 -12687.808} C_VEL
LIN {X 0,Y 367.604,Z 320.506,A -85,B 0,C 180,E1 -12688.904,E2 -12688.904} C_VEL
LIN {X 0,Y 367.588,Z 320.944,A -85,B 0,C 180,E1 -12690,E2 -12690} C_VEL
LIN {X 0,Y 367.583,Z 320.975,A -85,B 0,C 180,E1 -12691.095,E2 -12691.095} C_VEL
LIN {X 0,Y 367.526,Z 320.616,A -85,B 0,C 180,E1 -12692.191,E2 -12692.191} C_VEL
LIN {X 0,Y 367.445,Z 319.868,A -85,B 0,C 180,E1 -12693.289,E2 -12693.289} C_VEL
LIN {X 0,Y 367.462,Z 318.698,A -85,B 0,C 180,E1 -12694.387,E2 -12694.387} C_VEL
LIN {X 0,Y 367.457,Z 316.273,A -85,B 0,C 180,E1 -12695.981,E2 -12695.981} C_VEL
LIN {X 0,Y 367.661,Z 312.641,A -85,B 0,C 180,E1 -12697.689,E2 -12697.689} C_VEL
LIN {X 0,Y 367.981,Z 308.033,A -85,B 0,C 180,E1 -12699.342,E2 -12699.342} C_VEL
LIN {X 0,Y 368.683,Z 301.1,A -85,B 0,C 180,E1 -12701.267,E2 -12701.267} C_VEL
LIN {X 0,Y 369.678,Z 293.628,A -85,B 0,C 180,E1 -12702.907,E2 -12702.907} C_VEL
LIN {X 0,Y 370.697,Z 284.694,A -85,B 0,C 180,E1 -12704.495,E2 -12704.495} C_VEL
LIN {X 0,Y 371.911,Z 274.768,A -85,B 0,C 180,E1 -12705.902,E2 -12705.902} C_VEL
LIN {X 0,Y 373.239,Z 264.163,A -85,B 0,C 180,E1 -12707.11,E2 -12707.11} C_VEL
LIN {X 0,Y 374.438,Z 253.946,A -85,B 0,C 180,E1 -12708.04,E2 -12708.04} C_VEL
LIN {X 0,Y 375.619,Z 241.863,A -85,B 0,C 180,E1 -12708.9,E2 -12708.9} C_VEL
LIN {X 0,Y 376.691,Z 228.463,A -85,B 0,C 180,E1 -12709.587,E2 -12709.587} C_VEL
LIN {X 0,Y 377.402,Z 216.114,A -85,B 0,C 180,E1 -12710.009,E2 -12710.009} C_VEL
LIN {X 0,Y 378.7,Z 144.05,A -85,B 0,C 180,E1 -12711.434,E2 -12711.434} C_VEL
LIN {X 0,Y 375.693,Z 124.379,A -85,B 0,C 180,E1 -12712.056,E2 -12712.056} C_VEL
LIN {X 0,Y 372.248,Z 106.78,A -85,B 0,C 180,E1 -12712.704,E2 -12712.704} C_VEL
LIN {X 0,Y 373.96,Z 90.46,A -85,B 0,C 180,E1 -12716.208,E2 -12716.208} C_VEL
LIN {X 0,Y 373.533,Z 86.434,A -85,B 0,C 180,E1 -12717.153,E2 -12717.153} C_VEL
LIN {X 0,Y 371.2,Z 75.835,A -85,B 0,C 180,E1 -12719.8,E2 -12719.8} C_VEL
LIN {X 0,Y 368.94,Z 66.529,A -85,B 0,C 180,E1 -12722.302,E2 -12722.302} C_VEL
LIN {X 0,Y 368.928,Z 66.525,A -85,B 0,C 180,E1 -12725.001,E2 -12725.001} C_VEL
LIN {X 0,Y 368.909,Z 66.531,A -85,B 0,C 180,E1 -12728.64,E2 -12728.64} C_VEL
LIN {X 0,Y 368.88,Z 66.535,A -85,B 0,C 180,E1 -12732.009,E2 -12732.009} C_VEL
LIN {X 0,Y 368.878,Z 66.523,A -85,B 0,C 180,E1 -12735.175,E2 -12735.175} C_VEL
LIN {X 0,Y 368.908,Z 66.531,A -85,B 0,C 180,E1 -12738.181,E2 -12738.181} C_VEL
LIN {X 0,Y 368.912,Z 66.532,A -85,B 0,C 180,E1 -12741.358,E2 -12741.358} C_VEL
LIN {X 0,Y 368.935,Z 66.526,A -85,B 0,C 180,E1 -12745.146,E2 -12745.146} C_VEL
LIN {X 0,Y 368.926,Z 66.526,A -85,B 0,C 180,E1 -12749.046,E2 -12749.046} C_VEL
LIN {X 0,Y 368.977,Z 66.522,A -85,B 0,C 180,E1 -12751.564,E2 -12751.564} C_VEL
LIN {X 0,Y 368.997,Z 66.515,A -85,B 0,C 180,E1 -12754.02,E2 -12754.02} C_VEL
LIN {X 0,Y 368.931,Z 66.518,A -85,B 0,C 180,E1 -12757.605,E2 -12757.605} C_VEL
LIN {X 0,Y 368.987,Z 66.516,A -85,B 0,C 180,E1 -12761.108,E2 -12761.108} C_VEL
LIN {X 0,Y 368.995,Z 66.523,A -85,B 0,C 180,E1 -12764.535,E2 -12764.535} C_VEL
LIN {X 0,Y 369.003,Z 66.51,A -85,B 0,C 180,E1 -12767.907,E2 -12767.907} C_VEL
LIN {X 0,Y 369.185,Z 66.491,A -85,B 0,C 180,E1 -12771.846,E2 -12771.846} C_VEL
LIN {X 0,Y 369.139,Z 66.503,A -85,B 0,C 180,E1 -12774.538,E2 -12774.538} C_VEL
LIN {X 0,Y 369.314,Z 66.473,A -85,B 0,C 180,E1 -12777.819,E2 -12777.819} C_VEL
LIN {X 0,Y 369.454,Z 66.466,A -85,B 0,C 180,E1 -12780,E2 -12780} C_VEL
LIN {X 0,Y 369.314,Z 66.472,A -85,B 0,C 180,E1 -12782.181,E2 -12782.181} C_VEL
LIN {X 0,Y 369.183,Z 66.494,A -85,B 0,C 180,E1 -12786.572,E2 -12786.572} C_VEL
LIN {X 0,Y 369.061,Z 66.513,A -85,B 0,C 180,E1 -12789.869,E2 -12789.869} C_VEL
LIN {X 0,Y 369.035,Z 66.513,A -85,B 0,C 180,E1 -12793.773,E2 -12793.773} C_VEL
LIN {X 0,Y 368.988,Z 66.514,A -85,B 0,C 180,E1 -12797.743,E2 -12797.743} C_VEL
LIN {X 0,Y 368.908,Z 66.525,A -85,B 0,C 180,E1 -12801.221,E2 -12801.221} C_VEL
LIN {X 0,Y 368.937,Z 66.526,A -85,B 0,C 180,E1 -12804.777,E2 -12804.777} C_VEL
LIN {X 0,Y 368.929,Z 66.529,A -85,B 0,C 180,E1 -12808.441,E2 -12808.441} C_VEL
LIN {X 0,Y 368.909,Z 66.532,A -85,B 0,C 180,E1 -12810.988,E2 -12810.988} C_VEL
LIN {X 0,Y 368.935,Z 66.524,A -85,B 0,C 180,E1 -12814.854,E2 -12814.854} C_VEL
LIN {X 0,Y 368.877,Z 66.54,A -85,B 0,C 180,E1 -12818.635,E2 -12818.635} C_VEL
LIN {X 0,Y 368.872,Z 66.532,A -85,B 0,C 180,E1 -12822.008,E2 -12822.008} C_VEL
LIN {X 0,Y 368.878,Z 66.531,A -85,B 0,C 180,E1 -12825.176,E2 -12825.176} C_VEL
LIN {X 0,Y 368.869,Z 66.54,A -85,B 0,C 180,E1 -12828.176,E2 -12828.176} C_VEL
LIN {X 0,Y 368.895,Z 66.625,A -85,B 0,C 180,E1 -12831.604,E2 -12831.604} C_VEL
LIN {X 0,Y 370.171,Z 72.052,A -85,B 0,C 180,E1 -12833.2,E2 -12833.2} C_VEL
LIN {X 0,Y 378.619,Z 91.653,A -85,B 0,C 180,E1 -12834.262,E2 -12834.262} C_VEL
LIN {X 0,Y 379.69,Z 94.875,A -85,B 0,C 180,E1 -12834.408,E2 -12834.408} C_VEL
LIN {X 0,Y 378.063,Z 177.908,A -85,B 0,C 180,E1 -12836.035,E2 -12836.035} C_VEL
LIN {X 0,Y 377.464,Z 191.628,A -85,B 0,C 180,E1 -12836.524,E2 -12836.524} C_VEL
LIN {X 0,Y 376.863,Z 203.087,A -85,B 0,C 180,E1 -12837.136,E2 -12837.136} C_VEL
LIN {X 0,Y 375.966,Z 214.834,A -85,B 0,C 180,E1 -12837.967,E2 -12837.967} C_VEL
LIN {X 0,Y 374.871,Z 225.751,A -85,B 0,C 180,E1 -12838.965,E2 -12838.965} C_VEL
LIN {X 0,Y 373.582,Z 236.699,A -85,B 0,C 180,E1 -12840.229,E2 -12840.229} C_VEL
LIN {X 0,Y 372.491,Z 245.876,A -85,B 0,C 180,E1 -12841.55,E2 -12841.55} C_VEL
LIN {X 0,Y 371.415,Z 254.051,A -85,B 0,C 180,E1 -12842.991,E2 -12842.991} C_VEL
LIN {X 0,Y 370.254,Z 261.901,A -85,B 0,C 180,E1 -12844.718,E2 -12844.718} C_VEL
LIN {X 0,Y 369.413,Z 268.13,A -85,B 0,C 180,E1 -12846.452,E2 -12846.452} C_VEL
LIN {X 0,Y 368.763,Z 272.981,A -85,B 0,C 180,E1 -12848.184,E2 -12848.184} C_VEL
LIN {X 0,Y 368.282,Z 276.618,A -85,B 0,C 180,E1 -12849.91,E2 -12849.91} C_VEL
LIN {X 0,Y 367.978,Z 278.423,A -85,B 0,C 180,E1 -12851.054,E2 -12851.054} C_VEL
LIN {X 0,Y 367.663,Z 280.382,A -85,B 0,C 180,E1 -12852.897,E2 -12852.897} C_VEL
LIN {X 0,Y 367.504,Z 281.189,A -85,B 0,C 180,E1 -12854.471,E2 -12854.471} C_VEL
LIN {X 0,Y 367.481,Z 281.236,A -85,B 0,C 180,E1 -12855.604,E2 -12855.604} C_VEL
LIN {X 0,Y 367.518,Z 280.609,A -85,B 0,C 180,E1 -12857.233,E2 -12857.233} C_VEL
LIN {X 0,Y 367.571,Z 278.96,A -85,B 0,C 180,E1 -12858.978,E2 -12858.978} C_VEL
LIN {X 0,Y 367.763,Z 276.397,A -85,B 0,C 180,E1 -12860.652,E2 -12860.652} C_VEL
LIN {X 0,Y 368.034,Z 272.818,A -85,B 0,C 180,E1 -12862.319,E2 -12862.319} C_VEL
LIN {X 0,Y 368.366,Z 268.133,A -85,B 0,C 180,E1 -12863.977,E2 -12863.977} C_VEL
LIN {X 0,Y 368.928,Z 261.082,A -85,B 0,C 180,E1 -12865.904,E2 -12865.904} C_VEL
LIN {X 0,Y 369.589,Z 253.445,A -85,B 0,C 180,E1 -12867.548,E2 -12867.548} C_VEL
LIN {X 0,Y 370.438,Z 243.842,A -85,B 0,C 180,E1 -12869.185,E2 -12869.185} C_VEL
LIN {X 0,Y 371.342,Z 233.927,A -85,B 0,C 180,E1 -12870.543,E2 -12870.543} C_VEL
LIN {X 0,Y 372.218,Z 222.755,A -85,B 0,C 180,E1 -12871.759,E2 -12871.759} C_VEL
LIN {X 0,Y 373.03,Z 210.6,A -85,B 0,C 180,E1 -12872.795,E2 -12872.795} C_VEL
LIN {X 0,Y 373.618,Z 198.621,A -85,B 0,C 180,E1 -12873.573,E2 -12873.573} C_VEL
LIN {X 0,Y 374.042,Z 185.723,A -85,B 0,C 180,E1 -12874.168,E2 -12874.168} C_VEL
LIN {X 0,Y 374.401,Z 172.133,A -85,B 0,C 180,E1 -12874.557,E2 -12874.557} C_VEL
LIN {X 0,Y 375.501,Z 92.108,A -85,B 0,C 180,E1 -12876.089,E2 -12876.089} C_VEL
LIN {X 0,Y 374.118,Z 84.94,A -85,B 0,C 180,E1 -12876.295,E2 -12876.295} C_VEL
LIN {X 0,Y 372.755,Z 81.12,A -85,B 0,C 180,E1 -12876.436,E2 -12876.436} C_VEL
LIN {X 0,Y 369.476,Z 76.812,A -85,B 0,C 180,E1 -12876.679,E2 -12876.679} C_VEL
LIN {X 0,Y 364.749,Z 72.364,A -85,B 0,C 180,E1 -12877.076,E2 -12877.076} C_VEL
LIN {X 0,Y 362.891,Z 70.2,A -85,B 0,C 180,E1 -12877.43,E2 -12877.43} C_VEL
LIN {X 0,Y 362.513,Z 69.324,A -85,B 0,C 180,E1 -12877.64,E2 -12877.64} C_VEL
LIN {X 0,Y 362.163,Z 67.375,A -85,B 0,C 180,E1 -12878.232,E2 -12878.232} C_VEL
LIN {X 0,Y 361.966,Z 67.398,A -85,B 0,C 180,E1 -12882.333,E2 -12882.333} C_VEL
LIN {X 0,Y 361.967,Z 67.398,A -85,B 0,C 180,E1 -12884.621,E2 -12884.621} C_VEL
LIN {X 0,Y 361.965,Z 67.398,A -85,B 0,C 180,E1 -12888.099,E2 -12888.099} C_VEL
LIN {X 0,Y 361.867,Z 67.407,A -85,B 0,C 180,E1 -12891.655,E2 -12891.655} C_VEL
LIN {X 0,Y 361.932,Z 67.398,A -85,B 0,C 180,E1 -12895.29,E2 -12895.29} C_VEL
LIN {X 0,Y 361.913,Z 67.404,A -85,B 0,C 180,E1 -12897.779,E2 -12897.779} C_VEL
LIN {X 0,Y 361.843,Z 67.413,A -85,B 0,C 180,E1 -12901.629,E2 -12901.629} C_VEL
LIN {X 0,Y 361.879,Z 67.407,A -85,B 0,C 180,E1 -12905.345,E2 -12905.345} C_VEL
LIN {X 0,Y 361.875,Z 67.406,A -85,B 0,C 180,E1 -12909.027,E2 -12909.027} C_VEL
LIN {X 0,Y 361.84,Z 67.41,A -85,B 0,C 180,E1 -12912.829,E2 -12912.829} C_VEL
LIN {X 0,Y 361.838,Z 67.41,A -85,B 0,C 180,E1 -12915.944,E2 -12915.944} C_VEL
LIN {X 0,Y 361.839,Z 67.415,A -85,B 0,C 180,E1 -12919.244,E2 -12919.244} C_VEL
LIN {X 0,Y 361.867,Z 67.409,A -85,B 0,C 180,E1 -12922.777,E2 -12922.777} C_VEL
LIN {X 0,Y 361.858,Z 67.408,A -85,B 0,C 180,E1 -12925.719,E2 -12925.719} C_VEL
LIN {X 0,Y 361.876,Z 67.405,A -85,B 0,C 180,E1 -12929.672,E2 -12929.672} C_VEL
LIN {X 0,Y 361.957,Z 67.395,A -85,B 0,C 180,E1 -12933.475,E2 -12933.475} C_VEL
LIN {X 0,Y 361.895,Z 67.404,A -85,B 0,C 180,E1 -12937.145,E2 -12937.145} C_VEL
LIN {X 0,Y 361.91,Z 67.404,A -85,B 0,C 180,E1 -12940.723,E2 -12940.723} C_VEL
LIN {X 0,Y 361.936,Z 67.398,A -85,B 0,C 180,E1 -12943.066,E2 -12943.066} C_VEL
LIN {X 0,Y 362.002,Z 67.393,A -85,B 0,C 180,E1 -12946.528,E2 -12946.528} C_VEL
LIN {X 0,Y 362.034,Z 67.389,A -85,B 0,C 180,E1 -12949.938,E2 -12949.938} C_VEL
LIN {X 0,Y 362.164,Z 67.37,A -85,B 0,C 180,E1 -12953.313,E2 -12953.313} C_VEL
LIN {X 0,Y 362.282,Z 67.36,A -85,B 0,C 180,E1 -12957.776,E2 -12957.776} C_VEL
LIN {X 0,Y 362.428,Z 67.34,A -85,B 0,C 180,E1 -12960,E2 -12960} C_VEL
LIN {X 0,Y 362.282,Z 67.356,A -85,B 0,C 180,E1 -12962.223,E2 -12962.223} C_VEL
LIN {X 0,Y 362.15,Z 67.371,A -85,B 0,C 180,E1 -12966.686,E2 -12966.686} C_VEL
LIN {X 0,Y 362.002,Z 67.39,A -85,B 0,C 180,E1 -12970.063,E2 -12970.063} C_VEL
LIN {X 0,Y 362,Z 67.39,A -85,B 0,C 180,E1 -12973.899,E2 -12973.899} C_VEL
LIN {X 0,Y 361.969,Z 67.394,A -85,B 0,C 180,E1 -12977.938,E2 -12977.938} C_VEL
LIN {X 0,Y 361.863,Z 67.407,A -85,B 0,C 180,E1 -12981.655,E2 -12981.655} C_VEL
LIN {X 0,Y 361.928,Z 67.401,A -85,B 0,C 180,E1 -12985.29,E2 -12985.29} C_VEL
LIN {X 0,Y 361.916,Z 67.4,A -85,B 0,C 180,E1 -12987.778,E2 -12987.778} C_VEL
LIN {X 0,Y 361.848,Z 67.409,A -85,B 0,C 180,E1 -12991.285,E2 -12991.285} C_VEL
LIN {X 0,Y 361.856,Z 67.41,A -85,B 0,C 180,E1 -12994.28,E2 -12994.28} C_VEL
LIN {X 0,Y 361.864,Z 67.407,A -85,B 0,C 180,E1 -12997.223,E2 -12997.223} C_VEL
LIN {X 0,Y 361.837,Z 67.412,A -85,B 0,C 180,E1 -13000.755,E2 -13000.755} C_VEL
LIN {X 0,Y 361.819,Z 67.417,A -85,B 0,C 180,E1 -13004.368,E2 -13004.368} C_VEL
LIN {X 0,Y 361.838,Z 67.411,A -85,B 0,C 180,E1 -13007.568,E2 -13007.568} C_VEL
LIN {X 0,Y 361.871,Z 67.405,A -85,B 0,C 180,E1 -13010.973,E2 -13010.973} C_VEL
LIN {X 0,Y 361.876,Z 67.405,A -85,B 0,C 180,E1 -13014.655,E2 -13014.655} C_VEL
LIN {X 0,Y 361.84,Z 67.41,A -85,B 0,C 180,E1 -13018.37,E2 -13018.37} C_VEL
LIN {X 0,Y 361.908,Z 67.435,A -85,B 0,C 180,E1 -13020.126,E2 -13020.126} C_VEL
LIN {X 0,Y 364.272,Z 78.758,A -85,B 0,C 180,E1 -13022.777,E2 -13022.777} C_VEL
LIN {X 0,Y 365.195,Z 84.308,A -85,B 0,C 180,E1 -13024.036,E2 -13024.036} C_VEL
LIN {X 0,Y 364.534,Z 94.115,A -85,B 0,C 180,E1 -13026.117,E2 -13026.117} C_VEL
LIN {X 0,Y 363.476,Z 107.339,A -85,B 0,C 180,E1 -13028.894,E2 -13028.894} C_VEL
LIN {X 0,Y 368.166,Z 144.378,A -85,B 0,C 180,E1 -13029.866,E2 -13029.866} C_VEL
LIN {X 0,Y 367.072,Z 216.468,A -85,B 0,C 180,E1 -13031.295,E2 -13031.295} C_VEL
LIN {X 0,Y 366.523,Z 229.71,A -85,B 0,C 180,E1 -13031.772,E2 -13031.772} C_VEL
LIN {X 0,Y 365.654,Z 242.434,A -85,B 0,C 180,E1 -13032.451,E2 -13032.451} C_VEL
LIN {X 0,Y 364.827,Z 254.572,A -85,B 0,C 180,E1 -13033.348,E2 -13033.348} C_VEL
